	// final target position of joint4 in motor (not DH , same for below defination) 
	m_jnt4TargetPos: LREAL;
	
	// OTG for joint4 motion
	m_trajFilter :FB_secOrdTrajFilter;
	
	// command joint4 position and veloicty in motor for next cycle
	m_cmdJntPos: LREAL;
	m_cmdJntVel: LREAL;
	m_cmdJntAcc: LREAL;

	// PID for joint position
	m_jntPIDCtrl: FB_PID;
	m_jntCtrlTrq: LREAL;
	
END_VAR

METHOD PROTECTED calcJnt6Bias : LREAL
VAR_IN_OUT CONSTANT
	i_masterArm :FB_MasterArm;
END_VAR
IF 1= i_masterArm.armIdx THEN
	calcJnt6Bias :=i_masterArm.curJntPos[6]+PI/2;
ELSE 
	calcJnt6Bias := i_masterArm.curJntPos[6]-PI/2;
END_IF
END_METHOD

// calculate orientation manipulation velocity(in local coordinate)
METHOD calcManipVel : LREAL
VAR_IN_OUT CONSTANT
	i_masterArm :FB_MasterArm;
END_VAR
VAR
	wVelWrd,wVelLocal:Vec3d;
	rotT:Mat3d;
END_VAR
wVelWrd[1]:= i_masterArm.m_curCartLinkTwist[4];
wVelWrd[2]:= i_masterArm.m_curCartLinkTwist[5];
wVelWrd[3]:= i_masterArm.m_curCartLinkTwist[6];

matTranspose(i_masterArm.curCartPose.m_rot, rotT);
matMultiVec(rotT, wVelWrd, wVelLocal);

wVelLocal[3]:=0;
calcManipVel:=norm(wVelLocal);
END_METHOD

METHOD PROTECTED calcNullJaco : Mat4d;
VAR_IN_OUT CONSTANT
	i_masterArm :FB_MasterArm;
END_VAR
VAR
	i,j:INT;
	oriJaco:Mat34;
	oriJt:Mat43;
	oriJJt:Mat3d;
	oriJJtInv:Mat3d;
	oriJPinv:Mat43;
	JpinvJ :Mat4d;
	eye4d :Mat4d := g_eye4d;
END_VAR
// compute pinv of orientation jacobian
FOR i:=1 TO 3 DO
	FOR j:=1 TO 4 DO
		oriJaco[i,j]:=i_masterArm.simJaco[i+3,j+3];
	END_FOR
END_FOR
matTranspose(oriJaco, oriJt);
matMultiply(oriJaco ,oriJt , oriJJt);
invMat3(oriJJt, oriJJtInv);
matMultiply(oriJt, oriJJtInv, oriJPinv);

// calculate nullspace
matMultiply(oriJPinv, oriJaco, JpinvJ);
matSub(eye4d , JpinvJ, calcNullJaco);
END_METHOD

METHOD PROTECTED calcRedunPos : BOOL
VAR_IN_OUT CONSTANT
	i_masterArm :FB_MasterArm;
END_VAR

VAR 
	j6Bias :LREAL;
	curJntPos : Vec7d;
	jnt4LinkPos, jnt4TargetLinkPos :LREAL;
	singScale:LREAL;
END_VAR
// compute desired joint4 link position
// therotically should be link position, but joint controller use motor pos, so here also use motor pos, or will cause other problems
curJntPos :=  i_masterArm.curJntPos;
jnt4LinkPos:=i_masterArm.jnt4MotorToLink(curJntPos[2],curJntPos[3],curJntPos[4]);

// scale track motion near redundant singularity
IF ABS(m_oriNullJaco[1,1])<g_smallNum THEN
	singScale :=0;
ELSE
	singScale := MAX(ABS(m_oriNullJaco[2,1]/m_oriNullJaco[1,1]), ABS(m_oriNullJaco[3,1]/m_oriNullJaco[1,1]));
END_IF
j6Bias := m_jnt6Bias * ABS(singScale);

j6Bias := LIMIT (-m_maxTargetPosStep, j6Bias, m_maxTargetPosStep);
// final target position
jnt4TargetLinkPos := LIMIT(GVL_ArmJointParameters.g_minJntPos[i_masterArm.armIdx,4]+m_jntLimitBuffer, 
			jnt4LinkPos-j6Bias,GVL_ArmJointParameters.g_maxJntPos[i_masterArm.armIdx,4]-m_jntLimitBuffer); 
			
// convert from link position to motor position
m_jnt4TargetPos:=i_masterArm.jnt4LinkToMotor(curJntPos[2], curJntPos[3], jnt4TargetLinkPos);
END_METHOD

METHOD init : BOOL
VAR_IN_OUT CONSTANT
	i_masterArm :FB_MasterArm;
END_VAR
VAR
	currentRatioMotor2Jnt:LREAL;
END_VAR
m_cmdJntPos:=i_masterArm.curJntPos[4];
m_jnt4TargetPos:=m_cmdJntPos;
m_cmdJntVel:=0;

// init controller
currentRatioMotor2Jnt:=GVL_ArmJointParameters.g_motorTrqConst[4]*GVL_ArmJointParameters.g_motorReduction[4]/1000;
m_jntPIDCtrl.init(g_armCtrlCycleTime,m_redunJntKp,m_redunJntKd,m_redunJntKi,
		m_redunJntKiLimit* currentRatioMotor2Jnt,	m_redunJntCtrlLimit*currentRatioMotor2Jnt);

// init OTG
m_trajFilter.init(m_cmdJntPos,m_cmdJntVel,m_jnt4MaxFollowVel,m_jnt4MaxFollowAcc,g_armCtrlCycleTime);
END_METHOD

METHOD run : LREAL
VAR_IN_OUT CONSTANT
	i_masterArm :FB_MasterArm;
END_VAR
VAR_INPUT
	i_followEnable :BOOL;
END_VAR


VAR
	velScale,limitScale:LREAL;
	maxAcc, minDec:LREAL;
	wVel:Vec3d;

END_VAR
// joint 6 deviation from center
m_jnt6Bias := calcJnt6Bias(i_masterArm);

// calculate nullspace jacobian
m_oriNullJaco := calcNullJaco(i_masterArm);

// calculate manipulation angular velocity(exclude roll velocity)
m_curManipWVel := calcManipVel(i_masterArm);

// check if arm is static
m_trackFlag := startTrackCheck(i_masterArm);

// determin target position of joint4
IF i_followEnable THEN
	// update target redundant joint position
	IF  m_trackFlag THEN
		calcRedunPos(i_masterArm);
	ELSE
		// no control in static state
		IF ABS(m_cmdJntPos-m_jnt4TargetPos)< m_joint4TrackTol THEN
			m_jnt4TargetPos := i_masterArm.curJntPos[4];
			m_cmdJntPos :=i_masterArm.curJntPos[4];
			m_cmdJntVel:=0;
			m_jntPIDCtrl.reset();
			m_trajFilter.init(m_cmdJntPos,m_cmdJntVel,m_jnt4MaxFollowVel,m_jnt4MaxFollowAcc,g_armCtrlCycleTime);
		END_IF
	END_IF
END_IF

// scale following acceleration based on manipulation velocity
velScale := LIMIT (0,(ABS(m_curManipWVel)-m_jnt4MinAccVel)/(m_jnt4MaxAccVel-m_jnt4MinAccVel), 1.0);
maxAcc:=(m_jnt4MaxFollowAcc-m_jnt4MinFollowAcc)*velScale+m_jnt4MinFollowAcc;
//minDec:=m_trajFilter.minDec(m_jnt4TargetPos);
//maxAcc := MAX(maxAcc, minDec);

// scale acceleration when approaching limit
//m_accScaleNearLimit:=1;
limitScale := LIMIT(0.0,(ABS(m_jnt6Bias) - m_accScaleBiasLB)/(m_accScaleBiasUB-m_accScaleBiasLB),1.0);
m_accScaleNearLimit := 1+ limitScale * velScale * m_maxAccScaleNearLimit;
maxAcc:=maxAcc*m_accScaleNearLimit;


// run OTG
m_trajFilter.maxV:=m_curManipWVel;
m_trajFilter.maxA:=maxAcc;
m_trajFilter.run(m_jnt4TargetPos, 0.0, o_cmdAcc=>m_cmdJntAcc,o_cmdVel=>m_cmdJntVel, o_cmdPos=>m_cmdJntPos);

// joint position control torque control
m_jntCtrlTrq:=m_jntPIDCtrl.run(m_cmdJntPos,i_masterArm.curJntPos[4], m_cmdJntVel, i_masterArm.curJntVel[4]);

run:=m_jntCtrlTrq;
END_METHOD

METHOD startTrackCheck : BOOL
VAR_IN_OUT CONSTANT
	i_masterArm :FB_MasterArm;
END_VAR
IF (m_curManipWVel> m_staticVelThres AND i_masterArm.m_curLinkVel[6] * m_jnt6Bias > 0)  OR ABS(m_jnt6Bias)> m_staticBiasThres THEN
	startTrackCheck := TRUE;
ELSE
	startTrackCheck :=FALSE;
END_IF
END_METHOD

END_FUNCTION_BLOCK

// ---- FBs_TrajectoryPlanning/OTG/FB_secOrdTrajFilter.TcPOU
// reference: trajectory planning for automatic machines and robots
FUNCTION_BLOCK FB_secOrdTrajFilter
VAR_INPUT
END_VAR
VAR_OUTPUT
END_VAR
VAR
	// command pos and vel from last cycle
	m_cmdPos :LREAL;
	m_cmdVel :LREAL;
	
	// max velocity and acceleration
	m_maxV :LREAL;
	m_maxA :LREAL;
	
	// samping time
	m_Ts :LREAL;
	
	// middle variable
	ek,ek_dot,zk,zk_dot,m,sigma,satSigma :LREAL;

END_VAR

METHOD init : BOOL
VAR_INPUT
	i_curCmdPos : LREAL;
	i_curCmdVel :LREAL;
	i_maxV : LREAL;
	i_maxA :LREAL;
	i_Ts :LREAL;
END_VAR
m_cmdPos:=i_curCmdPos;
m_cmdVel:=i_curCmdVel;
m_maxV :=i_maxV;
m_maxA :=i_maxA;
m_Ts :=i_Ts;
END_METHOD

PROPERTY PUBLIC maxA : LREAL
GET
maxA:=m_maxA;
END_GET
SET
m_maxA :=maxA;
END_SET
END_PROPERTY

PROPERTY PUBLIC maxV : LREAL
GET
maxV:=m_maxV;
END_GET
SET
m_maxV:=maxV;
END_SET
END_PROPERTY

// get minimum deceleration to avoid overshoot
METHOD PUBLIC minDec : LREAL
VAR_INPUT
	i_targetPos : LREAL;
END_VAR

VAR
	dis : LREAL;
END_VAR
dis := i_targetPos-m_cmdPos;
// if target position reverse direciton, there always be a overshoot
IF dis*m_cmdVel <0 THEN
	minDec :=g_smallNum;
	RETURN;
END_IF

dis := MAX(g_smallNum, ABS(dis));
minDec := m_cmdVel *m_cmdVel /(2*dis);
END_METHOD

METHOD run : BOOL
VAR_INPUT
	i_targetPos, i_targetVel :LREAL;
END_VAR

VAR_OUTPUT
	o_cmdAcc, o_cmdVel, o_cmdPos :LREAL;
END_VAR
    ek:=(m_cmdPos-i_targetPos)/m_maxA;
    ek_dot:=(m_cmdVel-i_targetVel)/m_maxA;
    
    zk:=(ek/m_Ts+ek_dot/2)/m_Ts;
    zk_dot:=ek_dot/m_Ts;
    
    m:= floor((1+SQRT(1+8*ABS(zk)))/2);
    sigma:=zk_dot+zk/m+sign(zk)*(m-1)/2;
    satSigma:=MIN(1, MAX(-1,sigma));
    
    o_cmdAcc:=-m_maxA*satSigma*(1+sign(m_cmdVel*sign(sigma)+m_maxV-m_Ts*m_maxA))/2;
    o_cmdVel:=m_cmdVel+o_cmdAcc*m_Ts;
    o_cmdPos:=m_CmdPos+(o_cmdVel+m_cmdVel)*m_Ts/2;
	
	m_cmdVel := o_cmdVel;
	m_cmdPos := o_cmdPos;
END_METHOD

END_FUNCTION_BLOCK

// ---- AgiMaths/MatrixLib/invMat3.TcPOU
FUNCTION invMat3 : bool
VAR_IN_OUT CONSTANT
	mat :Mat3d;
END_VAR
VAR_IN_OUT
	invMat : Mat3d;
END_VAR
VAR
	n:INT:=3;
	m:INT:=1;
	b :ARRAY[1..3] OF LREAL := [3(0)];
	indxc,indxr, ipiv:ARRAY[1..3] OF INT := [3(0)];

	
	i,icol, irow, j,k,l,ll: INT;
	big, dum, pivinv,tmp: LREAL;
END_VAR

invMat := mat;
FOR i:=1 TO n DO   
    big:=0.0;
    FOR j:=1 TO n DO  
        IF (ipiv[j] <> 1) THEN
            FOR k:=1 TO n DO 
                IF (ipiv[k] = 0) THEN
                    IF (ABS(invMat[j,k]) >= big) THEN
                        big:=ABS(invMat[j,k]);
                        irow:=j;
                        icol:=k;
                    END_IF
                END_IF
            END_FOR
        END_IF
    END_FOR
    ipiv[icol]:=ipiv[icol]+1;
    
    IF (irow <> icol) THEN
        FOR l:=1 TO n DO 
            tmp:=invMat[irow,l];
            invMat[irow,l]:=invMat[icol,l];
            invMat[icol,l]:=tmp;
        END_FOR
 (*       FOR  l:=1 TO m DO  
            tmp:=b[irow,l];
            b[irow,l]:=b[icol,l];
            b[icol,l]:=tmp;
        END_FOR*)
    END_IF
	
    indxr[i]:=irow; 
    indxc[i]:=icol;
	
 	IF ABS(invMat[icol,icol]) < g_smallNum THEN  
          invMat3:=FALSE;
		  RETURN;
    END_IF
	
    pivinv:=1.0/invMat[icol,icol];
    invMat[icol,icol]:=1.0;
    FOR l:=1 TO n DO  
        invMat[icol,l] := invMat[icol,l]*pivinv;
    END_FOR
 (*   FOR l:=1 TO m DO 
        b[icol,l] := b[icol,l]*pivinv;
    END_FOR*)
    FOR ll:=1 TO n DO  
        IF (ll <> icol) THEN 
            dum:=invMat[ll,icol];
            invMat[ll,icol]:=0.0;
            FOR l:=1 TO n DO  
                invMat[ll,l]:=invMat[ll,l] - invMat[icol,l]*dum;
            END_FOR
   (*         FOR l:=1 TO m DO  
                b[ll,l]:=b[ll,l] - b[icol,l]*dum;
            END_FOR*)
        END_IF
    END_FOR

END_FOR


FOR l:=n-1 TO 1 BY -1 DO 
    IF (indxr[l] <> indxc[l]) THEN
        FOR k:=1 TO n DO
            tmp:=invMat[k,indxr[l]];
            invMat[k,indxr[l]]:=invMat[k,indxc[l]];
            invMat[k,indxc[l]]:=tmp;
        END_FOR
    END_IF
END_FOR

invMat3:=TRUE;

END_FUNCTION

// ---- AgiMaths/MatrixLib/matSub.TcPOU
// C = A - B;
FUNCTION matSub : BOOL
VAR_IN_OUT CONSTANT
	matA :ARRAY[*,*] OF LREAL;
	matB :ARRAY[*,*] OF LREAL;
END_VAR

VAR_IN_OUT 
	matC :ARRAY[*,*] OF LREAL;
END_VAR

VAR
	m,n :DINT;
	i,j, k :DINT;
 
END_VAR

m:=UPPER_BOUND(matC,1);
n:= UPPER_BOUND(matC,2);
ASSERT(UPPER_BOUND(matA,1)=m);
ASSERT(UPPER_BOUND(matA,2)=n);
ASSERT(UPPER_BOUND(matB,1)=m);
ASSERT(UPPER_BOUND(matB,2)=n);
FOR i:=1 TO m DO
	FOR j:=1 TO n DO
		matC[i,j]:=matA[i,j]-matB[i,j];
	END_FOR
END_FOR

END_FUNCTION

// ---- FBs_BasicControllers/FB_boundaryForceFeedback.TcPOU
FUNCTION_BLOCK FB_boundaryForceFeedback
VAR_INPUT
END_VAR
VAR_OUTPUT
END_VAR

VAR
	// force control parameters in local tip coordinate
//	m_oriKp :Vec3d :=[1, 1, 0.5];
//	m_oriKd :Vec3d :=[0.04,0.04, 0.01];
	m_oriKp :Vec3d :=[0.2, 0.2, 0.1];
	m_oriKd :Vec3d :=[0.02,0.02, 0.005];

	m_oriCartTrq,m_oriCartTrqLocal :Vec3d;
	
	m_posKp :LREAL := 200;
	m_posKd :LREAL := 10;
	m_posCartForce:Vec3d;
	
	
END_VAR

METHOD run : Vec7d

VAR_IN_OUT CONSTANT
	i_slaveIdx :INT;
	i_shoulderPose :ST_Frame;
	i_masterArm :FB_MasterArm;
	i_slaveStatus :ST_SlaveStatus;
END_VAR

VAR
	posErrInScope, oriErrInScope:Vec3d;
	posErr, oriErr:Vec3d;
	posErrLocal, oriErrLocal :Vec3d;
	vel, velLocal, wVel,wVelLocal :Vec3d;
	oriErrAxis, wVelProj :Vec3d;
	rotInv :Mat3d;
	oriJaco, oriJacoT :Mat3d;
	oriJntTrq :Vec3d;
	
	i,j:INT;
	posErrAxis, velProj :Vec3d;
	posJaco, posJacoT :Mat3d;
	posJntTrq :Vec3d;
	
	trqScale :LREAL;
END_VAR
run:=g_zeroVec7d;

FOR i:=1 TO 3 DO
	posErrInScope[i]:= -i_slaveStatus.m_masterSlavePoseError[i_slaveIdx][i];
	oriErrInScope[i]:= -i_slaveStatus.m_masterSlavePoseError[i_slaveIdx][i+3];
	vel[i]:=i_masterArm.curCartTwist[i];
	wVel[i]:=i_masterArm.curCartTwist[i+3];
END_FOR

// calculate pose error in shoulder coordinate
matTranspose(i_shoulderPose.m_rot, rotInv);
matMultiVec(rotInv, posErrInScope, posErr);
matMultiVec(rotInv, oriErrInScope, oriErr);
// ################### 	force  #########################
// add threshold
IF norm(posErr) > g_smallNum THEN
	// project error in tip coordinate
	matTranspose(i_masterArm.curCartPose.m_rot, rotInv);
	matMultiVec(rotInv, posErr, posErrLocal);
	matMultiVec(rotInv, oriErr, oriErrLocal);
	matMultiVec(rotInv, vel, velLocal);
	matMultiVec(rotInv, wVel, wVelLocal);
	
	// compute velocity in error direction
	posErrAxis := posErr;
	normalize(posErrAxis);
	vecMultiNum(posErrAxis, vecDot(vel, posErrAxis), velProj);
	
	// compute local cartesion torque
	FOR i:=1 TO 3 DO
		m_posCartForce[i]:= m_posKp * posErr[i]-m_posKd*velProj[i];
	END_FOR
	
	// compute joint space torque
	FOR i :=1 TO  3 DO
		FOR j:=1 TO 3 DO
			posJaco[i,j]:= i_masterArm.jaco[i,j];
		END_FOR
	END_FOR
	matTranspose(posJaco, posJacoT);
	matMultiVec(posJacoT, m_posCartForce, posJntTrq);
	
	// scale joint troque
	trqScale := 1;
	FOR i:=1 TO 3 DO 
		trqScale:=MAX(trqScale, ABS(posJntTrq[i]/GVL_ArmJointParameters.g_jntMaxTrq[i]));
	END_FOR
	
	run[1]:=posJntTrq[1]/trqScale;
	run[2]:=posJntTrq[2]/trqScale;
	run[3]:=posJntTrq[3]/trqScale;
END_IF


// ###################  torque #########################
// add threshold
IF norm(oriErr) > g_smallNum THEN
	// project error in tip coordinate
	matTranspose(i_masterArm.curCartPose.m_rot, rotInv);
	matMultiVec(rotInv, posErr, posErrLocal);
	matMultiVec(rotInv, oriErr, oriErrLocal);
	matMultiVec(rotInv, vel, velLocal);
	matMultiVec(rotInv, wVel, wVelLocal);
	
	// compute velocity in error direction
	oriErrAxis := oriErrLocal;
	normalize(oriErrAxis);
	vecMultiNum(oriErrAxis, vecDot(wVelLocal, oriErrAxis), wVelProj);
	
	// compute local cartesion torque
	FOR i:=1 TO 3 DO
		m_oriCartTrqLocal[i]:= m_oriKp[i] * oriErrLocal[i]-m_oriKd[i]*wVelProj[i];
	END_FOR
	
	// project torque back to shoulder coordinate
	matMultiVec(i_masterArm.curCartPose.m_rot, m_oriCartTrqLocal, m_oriCartTrq);
	
	// compute joint space torque
	// for simplicity, we current only use last 3 joint for torque feedback
	FOR i :=1 TO  3 DO
		FOR j:=1 TO 3 DO
			oriJaco[i,j]:= i_masterArm.jaco[i+3,j+4];
		END_FOR
	END_FOR
	matTranspose(oriJaco, oriJacoT);
	matMultiVec(oriJacoT, m_oriCartTrq, oriJntTrq);
	
	// scale joint troque
	trqScale := 1;
	FOR i:=1 TO 3 DO 
		trqScale:=MAX(trqScale, ABS(oriJntTrq[i]/GVL_ArmJointParameters.g_jntMaxTrq[i+4]));
	END_FOR
	
	run[5]:=oriJntTrq[1]/trqScale;
	run[6]:=oriJntTrq[2]/trqScale;
	run[7]:=oriJntTrq[3]/trqScale;
END_IF
END_METHOD

END_FUNCTION_BLOCK

// ---- AgiMaths/MatrixLib/vecDot.TcPOU
// vecB=VecA*num
FUNCTION vecDot : LREAL
VAR_IN_OUT CONSTANT
	vecA :ARRAY[*] OF LREAL;
	vecB :ARRAY[*] OF LREAL;
END_VAR

VAR
	m :DINT;
	i :DINT;
END_VAR

m:=UPPER_BOUND(vecA,1);
ASSERT(UPPER_BOUND(VecB,1)=m);

vecDot :=0;
FOR i:=1 TO m DO
	vecDot := vecDot + vecA[i]*vecB[i];
END_FOR

END_FUNCTION

// ---- AgiMaths/MatrixLib/vecSelfMultiNum.TcPOU
// vecA*=num
FUNCTION vecSelfMultiNum : BOOL
VAR_IN_OUT 
	vecA :ARRAY[*] OF LREAL;
END_VAR

VAR_INPUT
	num :LREAL;
END_VAR

VAR
	m :DINT;
	i :DINT;
 
END_VAR

m:=UPPER_BOUND(vecA,1);

FOR i:=1 TO m DO
		vecA[i]:=num*vecA[i];
END_FOR

END_FUNCTION

// ---- FBs_StateControllers/FB_StateCtrlClutch.TcPOU
// Brief: Master Arm Clutch
FUNCTION_BLOCK PUBLIC FB_StateCtrlClutch EXTENDS FB_MasterArmCtrlBase
VAR_INPUT
END_VAR
VAR_OUTPUT
END_VAR
VAR
	// orientation tracking parameters
	m_rotTrackKp : LREAL := 200;
	m_maxTrackVel :LREAL := PI;
	
	// redundant control parameters
	m_jnt4AdjustKp : LREAL :=10;
	m_jnt4MaxVel :LREAL :=pi/3 ;
	m_linearVelLb :LREAL := 0.02;
	m_linearVelUb :LREAL :=0.1;	
	
END_VAR

// override this function in each exact controller
METHOD PROTECTED calcCmdJntPos : BOOL

VAR_IN_OUT CONSTANT
	i_slaveIdx :INT;
	i_shoulderPose :ST_Frame;
	i_masterArm :FB_MasterArm;
	i_slaveStatus :ST_SlaveStatus;
END_VAR
var 
	i,j : INT;
	rotT,rotErr:Mat3d;
	angle : LREAL;
	axis,localAxis :Vec3d;
	oriJaco:Mat34;
	oriJt:Mat43;
	oriJJt:Mat3d;
	oriJJtInv:Mat3d;
	oriJPinv:Mat43;
	cartTrackVel:Vec3d;
	jntTrackVel:Vec4d;
	JpinvJ, nullJ:Mat4d;
	eye4d :Mat4d := g_eye4d;
	redunCtrlVel :Vec4d;
	jnt4TrackVel :LREAL;
	
END_VAR
// TODO: use matched slave arm orientation as target, 
//	and transform from view coordinate to arm coordinate 

// first three joints is passive control
FOR i:=1 TO 3 DO 
	m_cmdJntPos[i]:=i_masterArm.curJntPos[i];
	m_cmdJntVel[i]:=i_masterArm.curJntVel[i];
END_FOR

// compute cartesian tracking velocity
matTranspose(i_masterArm.simCartPose.m_rot, rotT);
matMultiply(rotT, m_cmdCartPose.m_rot, rotErr);
rot2AngAxis(rotErr, angle=>angle,axis=>localAxis);
matMultiVec(i_masterArm.simCartPose.m_rot, localAxis, axis);
vecMultiNum(axis, LIMIT(-m_maxTrackVel, angle*m_rotTrackKp, m_maxTrackVel), cartTrackVel);

// compute pinv of orientation jacobian
FOR i:=1 TO 3 DO
	FOR j:=1 TO 4 DO
		oriJaco[i,j]:=i_masterArm.simJaco[i+3,j+3];
	END_FOR
END_FOR
matTranspose(oriJaco, oriJt);
matMultiply(oriJaco ,oriJt , oriJJt);
invMat3(oriJJt, oriJJtInv);
matMultiply(oriJt, oriJJtInv, oriJPinv);
matMultiVec(oriJpinv, cartTrackVel, jntTrackVel);

// calculate nullspace
matMultiply(oriJPinv, oriJaco, JpinvJ);
matSub(eye4d , JpinvJ, nullJ);

// redundant velocity
jnt4TrackVel:=calcRedunVel(i_masterArm);
redunCtrlVel[1]:=nullJ[1,1]*jnt4TrackVel;
redunCtrlVel[2]:=nullJ[2,1]*jnt4TrackVel;
redunCtrlVel[3]:=nullJ[3,1]*jnt4TrackVel;
redunCtrlVel[4]:=nullJ[4,1]*jnt4TrackVel;

// update final command joint position and velocity
FOR i :=1 TO 4 DO 
//	m_cmdJntVel[i+3]:=jntTrackVel[i];
	m_cmdJntVel[i+3]:=jntTrackVel[i]+redunCtrlVel[i];
	m_cmdJntPos[i+3]:=m_cmdJntPos[i+3]+m_cmdJntVel[i+3]*g_armCtrlCycleTime;
END_FOR
END_METHOD

METHOD PROTECTED calcRedunVel : LREAL
VAR_IN_OUT CONSTANT
	i_masterArm :FB_MasterArm;
END_VAR

VAR 
	j6Bias,j5Bias :LREAL;
	velScale :LREAL;
	linearVel :Vec3d;
	curJntPos : Vec7d;
	jnt4LinkPos :LREAL;
END_VAR
// compute desired joint4 link position
curJntPos :=  i_masterArm.cmdJntPos;
jnt4LinkPos:=i_masterArm.jnt4MotorToLink(curJntPos[2],curJntPos[3],curJntPos[4]);
IF 1= i_masterArm.armIdx THEN
	j6Bias :=curJntPos[6]+PI/2;
ELSE 
	j6Bias := curJntPos[6]-PI/2;
END_IF

// scale based on joint5 position
j5Bias :=  LIMIT (0, ABS(curJntPos[5] -pi), pi/2);
j6Bias := j6Bias * ABS(COS(j5Bias));

// scale based on linear velocity
linearVel[1]:=i_masterArm.curCartTwist[1];
linearVel[2]:=i_masterArm.curCartTwist[2];
linearVel[3]:=i_masterArm.curCartTwist[3];
velScale :=LIMIT(0, (norm(linearVel)-m_linearVelLb)/(m_linearVelUb-m_linearVelLb),1.0);


calcRedunVel := LIMIT(-m_jnt4MaxVel, -j6Bias * m_jnt4AdjustKp * velScale ,m_jnt4MaxVel);

// joint limit
IF (calcRedunVel > 0 AND jnt4LinkPos+calcRedunVel * g_armCtrlCycleTime > GVL_ArmJointParameters.g_maxJntPos[i_masterArm.armIdx,4])
	 OR ( calcRedunVel <0 AND  jnt4LinkPos +calcRedunVel * g_armCtrlCycleTime< GVL_ArmJointParameters.g_minJntPos[i_masterArm.armIdx,4]) THEN
	 calcRedunVel :=0;
END_IF
END_METHOD

METHOD PUBLIC init : BOOL
VAR_IN_OUT CONSTANT
	i_masterArm	:FB_MasterArm;
END_VAR
VAR_IN_OUT 
	r_masterArmCtrlCmd :ST_ArmCtrlCmds;
END_VAR

VAR
	i:INT;
END_VAR
SUPER^.Init(i_masterArm,r_masterArmCtrlCmd);

m_jntOPMode[1] := DriverOPMode_Trq;
m_jntOPMode[2] := DriverOPMode_Trq;
m_jntOPMode[3] := DriverOPMode_Trq;
m_jntOPMode[4] := DriverOPMode_PosTrq;
m_jntOPMode[5] := DriverOPMode_PosTrq;
m_jntOPMode[6] := DriverOPMode_PosTrq;
m_jntOPMode[7] := DriverOPMode_PosTrq;

// update commands to arm
copyCmds(r_masterArmCtrlCmd);
END_METHOD

END_FUNCTION_BLOCK

// ---- FBs_StateControllers/FB_StateCtrlEndoscope.TcPOU
// Brief: Master Arm Endoscope Control
FUNCTION_BLOCK PUBLIC FB_StateCtrlEndoscope EXTENDS FB_MasterArmCtrlBase
VAR_INPUT
END_VAR
VAR_OUTPUT
END_VAR
VAR
	// enter endoscope control for the first time
	m_firstIn :BOOL := TRUE;
	
	//arm force control in base coordinate
	m_impCtrlInBase:BOOL;
	
	// force control parameters in base coordinate
	m_kpBase:Vec6d:=[1,1,1,1,1,1];
	m_kdBase:Vec6d:=[0.01,0.01,0.01,0.01,0.01,0.01];
	
	//endoscope motion scale
	m_endoMotionScale:LREAL:=1;
	
	// force control parameters in tcp coordinate
	m_kpTcp:Vec6d:=[100,100,100,1,1,0.5];
	m_kdTcp:Vec6d:=[1,1,1,0.04,0.04,0.01]; //[5,5,5,0.04,0.04,0.01];
	
	//joint 6 KP/KD
	m_Kp6:LREAL:=1.0; //1
	m_Kd6:LREAL:=0.01; //0.01
	
	//expected joint 6 position
	m_ExpJ6Pos:LREAL;
	
	//time
	m_t:LREAL;	
END_VAR

// override this function in each exact controller
METHOD PROTECTED calcCmdJntPos : BOOL

VAR_IN_OUT CONSTANT
	i_slaveIdx :INT;
	i_shoulderPose :ST_Frame;
	i_masterArm :FB_MasterArm;
	i_slaveStatus :ST_SlaveStatus;
END_VAR
VAR 

END_VAR
m_cmdJntPos:=i_masterArm.curJntPos;
m_cmdJntVel:=i_masterArm.curJntVel;
m_cmdCartPose:=i_masterArm.curCartPose;
END_METHOD

// override this function in each exact controller
METHOD PROTECTED calcCmdJntTrq : BOOL

VAR_IN_OUT CONSTANT
	i_slaveIdx :INT;
	i_shoulderPose :ST_Frame;
	i_masterArm :FB_MasterArm;
	i_slaveStatus :ST_SlaveStatus;
END_VAR

VAR	
	i:INT;
	
	//position variables
	masterPos,slavePos:ST_Frame;
	masterPosFirst,slavePosFirst:ST_Frame;
	ArmTarPos:ST_Frame;
	posInc:Vec3d;		
	tmpMat3d : Mat3d;
	rotInv:Mat3d;
	
	//velocity variables
	vel, velLocal, wVel,wVelLocal :Vec3d;
	spatialVel,spatialVelInTcp:Vec6d;
	
	//force variables
	spatialForceP1,spatialForceP2:Vec3d;	
	spatialForceP1Base,spatialForceP2Base:Vec3d;		
	spatialForTcp,spatialForBase,spatialForTemp:Vec7d;
	
	//joint torque variables
	simJaco:Mat67;
	JacoT :Mat76;	
	jntTorVec:Vec7d;
	dynaNullspace:Mat7d;	
	TorqueNullSpace:Vec7d; //joint torque for null space
	jntOptTor:LREAL; //joint 6 optimization torque
	jntTorqueSum:Vec7d;		
	jntImpTor:Vec7d;
	
	//master arm posture error variables
	posErr,posErrInBase,posErrInTcp:Vec3d;
	rotErr :Mat3d;
	errAngle : LREAL;
	errAxisLocal, errAxis,errAxis2,errAxisInBase,errAxisInTcp :Vec3d;
	masterPoseError,masterPoseErrorInTcp :Vec6d;
END_VAR

//determine slave arm space position relative to endoscope
masterPos:=transform(i_shoulderPose,i_masterArm.simCartPose);
slavePos:=i_slaveStatus.m_curArmPose[i_slaveIdx];

//system parameters initial
IF (m_firstIn=TRUE) THEN
	m_firstIn:=FALSE;
	masterPosFirst:=masterPos;
	slavePosFirst:=slavePos;	
	m_ExpJ6Pos:=i_masterArm.curJntPos[6];	
END_IF

m_t:=m_t+g_armCtrlCycleTime;
IF (m_t<=0.050) THEN
	m_firstIn:=TRUE;
	RETURN;	
END_IF




//calculating slave arm position incresement，and determine master arm space position and posture
vecSub(slavePos.m_pos,slavePosFirst.m_pos,posInc);
vecMultiNum(posInc,1.0/m_endoMotionScale,posInc);
vecAdd(posInc,masterPosFirst.m_pos,ArmTarPos.m_pos);
ArmTarPos.m_rot:=slavePos.m_rot;



//calculating master arm position error and postrue error
vecSub(ArmTarPos.m_pos, masterPos.m_pos, PosErr);
matTranspose(masterPos.m_rot, tmpMat3d);
matMultiply(tmpMat3d, ArmTarPos.m_rot, rotErr);
rot2AngAxis(rotErr, angle=>errAngle, axis=>errAxisLocal);
matMultiVec(masterPos.m_rot, errAxisLocal, errAxis);



//transform the error to arm base coordinate
matTranspose(i_shoulderPose.m_rot,tmpMat3d); //transform matrix from eye to base
matMultiVec(tmpMat3d, PosErr,posErrInBase);
matMultiVec(tmpMat3d, errAxis,errAxis2);
vecMultiNum(errAxis2,errAngle,errAxisInBase);
FOR i:=1 TO 3 BY 1 DO
	masterPoseError[i]:=posErrInBase[i];
	masterPoseError[i+3]:=errAxisInBase[i];
END_FOR



//transform the error to TCP coordinate
matTranspose(i_masterArm.curCartPose.m_rot, rotInv);
matMultiVec(rotInv, posErrInBase, posErrInTcp);
matMultiVec(rotInv, errAxisInBase, errAxisInTcp);
FOR i:=1 TO 3 BY 1 DO
	masterPoseErrorInTcp[i]:=posErrInTcp[i];
	masterPoseErrorInTcp[i+3]:=errAxisInTcp[i];
END_FOR



//determine master arm space velocity in base coordinate
FOR i:=1 TO 3 DO
	vel[i]:=i_masterArm.curCartTwist[i];
	wVel[i]:=i_masterArm.curCartTwist[i+3];
	spatialVel[i]:=vel[i];
	spatialVel[i+3]:=wVel[i];
END_FOR



//transform master arm space velocity to tcp coordinate
matMultiVec(rotInv, vel, velLocal);
matMultiVec(rotInv, wVel, wVelLocal);
FOR i:=1 TO 3 DO
	spatialVelInTcp[i]:=velLocal[i];
	spatialVelInTcp[i+3]:=wVelLocal[i];
END_FOR



//Jacobian matrix
simJaco:=i_masterArm.Jaco;



//Based on the above pose deviation values, input them into the impedance control equation and derive the impedance joint torque value
IF (m_impCtrlInBase=TRUE) THEN
	FOR i:=1 TO 6 BY 1 DO
		spatialForBase[i]:=m_kpBase[i]*masterPoseError[i]-m_kdBase[i]*spatialVel[i]; //(-1)*err*(-1)=err
	END_FOR
	matMultiVec(i_masterArm.m_lambda, spatialForBase, spatialForTemp);
	matTranspose(simJaco,JacoT);
	matMultiVec(JacoT, spatialForTemp, jntImpTor);	
	
ELSE // impedance control in tcp coordinate
	FOR i:=1 TO 6 BY 1 DO
		spatialForTcp[i]:=m_kpTcp[i]*masterPoseErrorInTcp[i]-m_kdTcp[i]*spatialVelInTcp[i];
	END_FOR
	
	//Splitting spatial forces into two parts
	FOR i:=1 TO 3 BY 1 DO
		spatialForceP1[i]:=spatialForTcp[i];
		spatialForceP2[i]:=spatialForTcp[i+3];
	END_FOR
	
	// project torque back to base coordinate	
	matMultiVec(i_masterArm.curCartPose.m_rot, spatialForceP1, spatialForceP1Base);	
	matMultiVec(i_masterArm.curCartPose.m_rot, spatialForceP2, spatialForceP2Base);	
	
	FOR i:=1 TO 3 BY 1 DO
		spatialForBase[i]:=spatialForceP1Base[i];
		spatialForBase[i+3]:=spatialForceP2Base[i];
	END_FOR
	
	//compute joint space torque
	matTranspose(simJaco,JacoT);
	matMultiVec(JacoT, spatialForBase, jntImpTor);	
END_IF




//To ensure that joint 6 is in the appropriate position, a single joint impedance controller is constructed
jntOptTor:=m_Kp6*(m_ExpJ6Pos-i_masterArm.curJntPos[6])-m_Kd6*i_masterArm.curJntVel[6];
(*
//Project the torque of joint 6 onto null space
jntTorVec[6]:=jntOptTor;
dynaNullspace:=i_masterArm.dynaNullspace;
matMultiVec(dynaNullspace, jntTorVec, TorqueNullSpace);	

//Calculate the sum of impedance control torque and zero space torque
vecAdd(jntImpTor,TorqueNullSpace,jntTorqueSum);
m_cmdJntTrq:=jntTorqueSum;
*)
m_cmdJntTrq:=jntImpTor;
m_cmdJntTrq[6]:=jntOptTor;
END_METHOD

// override this function in each exact controller
// NOTICE: set joint control mode here, and do some initialization if needed
METHOD PUBLIC init : BOOL
VAR_IN_OUT CONSTANT
	i_masterArm	:FB_MasterArm;
END_VAR
VAR_IN_OUT 
	r_masterArmCtrlCmd :ST_ArmCtrlCmds;
END_VAR

SUPER^.Init(i_masterArm,r_masterArmCtrlCmd);

m_jntOPMode[1] := DriverOPMode_Trq;
m_jntOPMode[2] := DriverOPMode_Trq;
m_jntOPMode[3] := DriverOPMode_Trq;
m_jntOPMode[4] := DriverOPMode_Trq;
m_jntOPMode[5] := DriverOPMode_Trq;
m_jntOPMode[6] := DriverOPMode_Trq;
m_jntOPMode[7] := DriverOPMode_Trq;

m_firstIn:=TRUE;
m_t:=0;

// update commands to arm
copyCmds(r_masterArmCtrlCmd);
END_METHOD

METHOD relativeAngle : bool
VAR_INPUT
	armId:INT;
	x:LREAL;
	y:LREAL;
END_VAR

VAR_OUTPUT
	angle:LREAL;
END_VAR

VAR
	
END_VAR


angle:=atan2(y,x);
IF (armId=1) AND (angle<0) THEN
	angle:=angle+2*pi;
END_IF
END_METHOD

END_FUNCTION_BLOCK

// ---- AgiMaths/Frames/transform.TcPOU
FUNCTION transform : ST_Frame
VAR_IN_OUT CONSTANT
	i_frame1 :ST_Frame;
	i_frame2 :ST_Frame;
END_VAR
VAR
END_VAR

matMultiply(i_frame1.m_rot, i_frame2.m_rot, transform.m_rot);
matMultiVec(i_frame1.m_rot, i_frame2.m_pos,transform.m_pos );
vecAdd(transform.m_pos,i_frame1.m_pos,transform.m_pos);

END_FUNCTION

// ---- FBs_StateControllers/FB_StateCtrlCart.TcPOU
// Brief: Master Arm Cart Control
FUNCTION_BLOCK PUBLIC FB_StateCtrlCart EXTENDS FB_MasterArmCtrlBase
VAR_INPUT
END_VAR
VAR_OUTPUT
END_VAR
VAR
END_VAR

METHOD PUBLIC init : BOOL
VAR_IN_OUT CONSTANT
	i_masterArm	:FB_MasterArm;
END_VAR
VAR_IN_OUT 
	r_masterArmCtrlCmd :ST_ArmCtrlCmds;
END_VAR
// check if to hold the command joint position unchanged
m_holdLastCmds := checkToHoldLastCmds(i_masterArm);

// init
SUPER^.Init(i_masterArm,r_masterArmCtrlCmd);
END_METHOD

END_FUNCTION_BLOCK

// ---- FBs_StateControllers/FB_StateCtrlGraCali.TcPOU
// Brief: Master Arm Home Posture
FUNCTION_BLOCK PUBLIC FB_StateCtrlGraCali EXTENDS FB_MasterArmCtrlBase
VAR_INPUT
END_VAR
VAR_OUTPUT
END_VAR
VAR CONSTANT
	m_caliMotionSegs :INT :=6;	
END_VAR
VAR
	// cali trajectory
	m_leftGraCaliTraj :ARRAY [1..m_caliMotionSegs, 1..g_mJntNum] OF LREAL:=
		// first calibration traj
		[0,  -60*g_deg2Rad,    0.0,  -195*g_deg2Rad,  270*g_deg2rad,  -60*g_deg2rad, 0.0 , 
		 0, -120*g_deg2rad,   0.0,  -165*g_deg2rad,   90*g_deg2rad,  -120*g_deg2rad,  0,
		 0,  -60*g_deg2Rad,    0.0,  -195*g_deg2Rad,  270*g_deg2rad,  -60*g_deg2rad, 0.0 , 
		// second calibration traj
		 0.0,  -75*g_deg2Rad,   30*g_deg2Rad,  -195*g_deg2Rad,  180*g_deg2Rad,  -90*g_deg2Rad,    0,
		 0.0,  -105*g_deg2Rad,  -30*g_deg2Rad, -165*g_deg2Rad,  180*g_deg2Rad,  -90*g_deg2Rad,     0,
		0.0,  -75*g_deg2Rad,   30*g_deg2Rad,  -195*g_deg2Rad,  180*g_deg2Rad,  -90*g_deg2Rad,    0];
		
	m_rightGraCaliTraj :ARRAY [1..m_caliMotionSegs, 1..g_mJntNum] OF LREAL:=
		// first calibration traj
		[0,   -60*g_deg2Rad,    0.0,   75*g_deg2Rad,   90*g_deg2Rad,   60*g_deg2Rad,  0.0,
		 0.0,  -120*g_deg2Rad,  0.0,  -75*g_deg2Rad,  270*g_deg2Rad,  120*g_deg2Rad,  0.0,
		 0,   -60*g_deg2Rad,    0.0,   75*g_deg2Rad,   90*g_deg2Rad,   60*g_deg2Rad,  0.0,
		// second calibration traj
		 0.0,  -75*g_deg2Rad,   30*g_deg2Rad,  -15*g_deg2Rad,  180*g_deg2Rad,   90*g_deg2Rad,    0,
		 0.0, -105*g_deg2Rad,  -30*g_deg2Rad,   15*g_deg2Rad,  180*g_deg2Rad,   90*g_deg2Rad,    0,
		 0.0,  -75*g_deg2Rad,   30*g_deg2Rad,  -15*g_deg2Rad,  180*g_deg2Rad,   90*g_deg2Rad,    0];
	

	m_transMaxjntVel:Vec7d:=[7(30*g_deg2rad)];
	m_caliMaxjntVel:Vec7d:=[7(3.0*g_deg2rad)];
	m_caliMaxjntAcc:Vec7d:=[7(1.0)];
	m_caliMaxjntJerk:Vec7d:=[7(2.0)];
	
	m_caliTrajIdx: INT := 1;
	m_caliPlanner: ARRAY[1..m_caliMotionSegs] OF FB_TrajMoveJ;
	
	
END_VAR

// override this function in each exact controller
METHOD PROTECTED calcCmdJntPos : BOOL

VAR_IN_OUT CONSTANT
	i_slaveIdx :INT;
	i_shoulderPose :ST_Frame;
	i_masterArm :FB_MasterArm;
	i_slaveStatus :ST_SlaveStatus;
END_VAR
VAR 
	i :INT;
	curJntVel :Vec7d;
END_VAR
// check if planner is ready
IF m_caliPlanner[m_caliTrajIdx].isGene = FALSE THEN
	calcCmdJntPos:=FALSE;
	RETURN;
END_IF

// traj plan
calcCmdJntPos :=m_caliPlanner[m_caliTrajIdx].evaluate(m_timePeriod, jntPos=> m_cmdJntPos, jntVel=>m_cmdJntVel, jntAcc=> m_cmdJntAcc);

// check if to transit to next segment
curJntVel :=i_masterArm.curJntVel;
IF(m_timePeriod > m_caliPlanner[m_caliTrajIdx].duration  AND norm(curJntVel)<7*g_jntStaticVelThres) THEN
	m_caliTrajIdx:=m_caliTrajIdx+1;
	m_timePeriod:=0;
END_IF

// check if to terminated
IF(m_caliTrajIdx > m_caliMotionSegs) THEN
	m_isFinished:=TRUE;
END_IF
END_METHOD

METHOD PUBLIC init : BOOL
VAR_IN_OUT CONSTANT
	i_masterArm	:FB_MasterArm;
END_VAR
VAR_IN_OUT 
	r_masterArmCtrlCmd :ST_ArmCtrlCmds;
END_VAR

VAR
	i,j :INT;
	startJntPos,endJntPos ,maxVel :Vec7d;
	
	
	
END_VAR
SUPER^.Init(i_masterArm,r_masterArmCtrlCmd);
m_caliTrajIdx :=1;

FOR i:=1 TO m_caliMotionSegs DO
	IF i=1 OR i = 4 THEN
		maxVel := m_transMaxjntVel;
	ELSE
		maxVel := m_caliMaxjntVel;
	END_IF
	
	IF i_masterArm.armIdx=1 THEN
		FOR j:=1 TO 7 DO 
			endJntPos[j]:=m_leftGraCaliTraj[i,j];
			IF i =1 THEN
				startJntPos[j]:=i_masterArm.curJntPos[j];
			ELSE
				startJntPos[j]:=m_leftGraCaliTraj[i-1,j];
			END_IF
		END_FOR
	ELSE
		FOR j:=1 TO 7 DO 
			endJntPos[j]:=m_rightGraCaliTraj[i,j];
			IF i =1 THEN
				startJntPos[j]:=i_masterArm.curJntPos[j];
			ELSE
				startJntPos[j]:=m_rightGraCaliTraj[i-1,j];
			END_IF
		END_FOR
	END_IF
	
	m_caliPlanner[i].init(startJntPos,endJntPos,maxVel, m_caliMaxJntAcc, m_caliMaxJntAcc);
END_FOR


// update commands to arm
copyCmds(r_masterArmCtrlCmd);
END_METHOD

END_FUNCTION_BLOCK

// ---- FBs_StateControllers/FB_StateCtrlTest.TcPOU
// Brief: Master Arm Test
FUNCTION_BLOCK PUBLIC FB_StateCtrlTest EXTENDS FB_MasterArmCtrlBase
VAR_INPUT
END_VAR
VAR_OUTPUT
END_VAR
VAR
	// ################ variables for single DH  joint test ##################
	m_freqTestFlag :BOOL:=FALSE;
	m_initJntPos :Vec7d;
	m_jntMotionFreq :Vec7d :=[0.2, 0.2, 0.1, 4(0.1)];
	m_jntMotionRange :Vec7d :=[pi/6, pi/6, 0.1, 4(pi/6)];
	m_testJntIdx :INT :=1;
	
	m_stepTestFlag :BOOL :=FALSE;
	m_jntStep : LREAL := 5*g_deg2Rad;
	
END_VAR

METHOD PROTECTED calcCmdJntPos : BOOL
VAR_IN_OUT CONSTANT
	i_slaveIdx :INT;
	i_shoulderPose :ST_Frame;
	i_masterArm :FB_MasterArm;
	i_slaveStatus :ST_SlaveStatus;
END_VAR

VAR 
	i:INT :=0;
	errThres :LREAL;
	m_masterGripAngle: INT;
END_VAR
// Just for joint controller test
IF m_testJntIdx >=1 AND m_testJntIdx <=7 THEN
	IF m_freqTestFlag THEN 
		m_cmdJntPos[m_testJntIdx]:=m_initJntPos[m_testJntIdx]+m_jntMotionRange[m_testJntIdx]/2
										+0.5*m_jntMotionRange[m_testJntIdx]*SIN(2*pi*m_jntMotionFreq[m_testJntIdx]*m_timePeriod-pi/2);
		m_cmdJntVel[m_testJntIdx]:=0.5*m_jntMotionRange[m_testJntIdx]*2*pi*m_jntMotionFreq[m_testJntIdx]*COS(2*pi*m_jntMotionFreq[m_testJntIdx]*m_timePeriod-pi/2);
	ELSIF m_stepTestFlag THEN
		m_cmdJntPos[m_testJntIdx]:=m_initJntPos[m_testJntIdx]+m_jntStep;
		m_cmdJntVel[m_testJntIdx]:=0;
	ELSE
		m_timePeriod:=0;
	END_IF
	
END_IF


FOR i:=1 TO 3 DO 
		errThres :=5*g_deg2rad;
	IF ABS(m_cmdJntPos[i]-i_masterArm.curJntPos[i])>errThres THEN
		m_isFinished:=TRUE;
	END_IF
	
END_FOR
END_METHOD

METHOD PUBLIC init : BOOL
VAR_IN_OUT CONSTANT
	i_masterArm	:FB_MasterArm;
END_VAR
VAR_IN_OUT 
	r_masterArmCtrlCmd :ST_ArmCtrlCmds;
END_VAR
// check if to hold the command joint position unchanged
m_holdLastCmds := checkToHoldLastCmds(i_masterArm);

// init
SUPER^.Init(i_masterArm,r_masterArmCtrlCmd);

m_initJntPos := i_masterArm.curJntPos;

// update commands to arm
copyCmds(r_masterArmCtrlCmd);
END_METHOD

END_FUNCTION_BLOCK

// ---- FBs_StateControllers/FB_StateCtrlDisable.TcPOU
// Brief: Master Arm Error Hold
FUNCTION_BLOCK PUBLIC FB_StateCtrlDisable EXTENDS FB_MasterArmCtrlBase
VAR_INPUT
END_VAR
VAR_OUTPUT
END_VAR
VAR
END_VAR

// override this function in each exact controller
METHOD PROTECTED calcCmdJntPos : BOOL

VAR_IN_OUT CONSTANT
	i_slaveIdx :INT;
	i_shoulderPose :ST_Frame;
	i_masterArm :FB_MasterArm;
	i_slaveStatus :ST_SlaveStatus;
END_VAR
var 
	i,j : INT;

	
END_VAR
m_cmdJntPos:= i_masterArm.curJntPos;
m_cmdJntVel := g_zeroVec7d;
END_METHOD

METHOD PUBLIC init : BOOL
VAR_IN_OUT CONSTANT
	i_masterArm	:FB_MasterArm;
END_VAR
VAR_IN_OUT 
	r_masterArmCtrlCmd :ST_ArmCtrlCmds;
END_VAR

VAR
	i:INT;
END_VAR
SUPER^.Init(i_masterArm,r_masterArmCtrlCmd);

// disable all joints
m_jntEnableFlag :=g_zeroVec7i;
END_METHOD

END_FUNCTION_BLOCK

// ---- FBs_StateControllers/FB_StateCtrlPerformance.TcPOU
FUNCTION_BLOCK FB_StateCtrlPerformance EXTENDS FB_MasterArmCtrlBase
VAR_INPUT
END_VAR
VAR_OUTPUT
END_VAR
VAR CONSTANT
	//max number of data recording points
	m_dataSum:INT:=8000;
END_VAR

VAR
	//test step
	m_testStep:INT:=-1;
	
	//test joint
	m_testJnt:INT;
	
	//Extreme joint position
	m_minJntPos: ARRAY[1..g_mJntNum] OF LREAL;
	m_maxJntPos: ARRAY[1..g_mJntNum] OF LREAL;
	
	//home position
	m_homeJntPos:ARRAY[1..g_mJntNum] OF LREAL;
	
	//Joint motion speed, acceleration, and jerk
	m_caliMaxjntVel:Vec7d:=[7(3.0*g_deg2rad)];
	m_caliMaxjntAcc:Vec7d:=[7(1.0)];
	m_caliMaxjntJerk:Vec7d:=[7(2.0)];
	
	//arm parameters
	m_armId:INT;
	
	//index
	i,j,id,idx:INT;
	
	//trajectory planner
	m_caliTrajIdx: INT := 1;
	m_jntIdx:INT:=1;
	m_caliMotionSegs :INT :=4;
	m_caliPlanner: ARRAY[1..7,1..g_mJntNum] OF FB_TrajMoveJ;
	m_caliPlannerStart: FB_TrajMoveJ;
	
	//speed test variable
	m_speedMaxTest:BOOL;
	
	//sampling interval
	m_samplingInterval:INT:=80;
	
	//Number of data records
	m_dataRecordNum_2,m_dataRecordNum_3:ARRAY[1..g_mJntNum] OF INT;
			
	//The current values of the second and third trajectories
	m_jntCurrentId2:ARRAY[1..m_dataSum,1..g_mJntNum] OF LREAL;
	m_jntCurrentId3:ARRAY[1..m_dataSum,1..g_mJntNum] OF LREAL;
	
	//friction record value
	m_CoulombFriction,m_ViscousFriction:ARRAY[1..m_dataSum,1..g_mJntNum] OF LREAL;
	
	//friction summation
	m_CoulombFrictionSum,m_ViscousFrictionSum:ARRAY[1..g_mJntNum] OF LREAL;
	
	//friction averange
	m_CoulombFrictionAve,m_ViscousFrictionAve:ARRAY[1..g_mJntNum] OF LREAL;
	
	//friction maxmum value
	m_CoulombFrictionMax,m_ViscousFrictionMax:ARRAY[1..g_mJntNum] OF LREAL;
	
	//Dynamic performance testing time
	m_t:LREAL;
	
	//Dynamic performance testing motion range
	m_motionRange:ARRAY[1..g_mJntNum] OF LREAL:=[0.1,0.1,0.1,0.1,0.1,0.1,0.1];
	
	//Starting point for dynamic performance testing
	m_posOffset:ARRAY[1..g_mJntNum] OF LREAL;
	
	//Number of dynamic performance tests
	m_testNum:INT:=5;
	
	//motion Frequency and angular frequency
	//m_Frequency:LREAL:=3; 	m_w:LREAL;
	m_Frequency:LREAL:=1; 	m_w:LREAL;
	
	//motion Frequency and angular frequency for speed test
	m_FrequencySpeed:LREAL:=0.5; 	m_wSpeed:LREAL;
	
	//motion range for maximum speed test
	//m_motionRangeSpeed:ARRAY[1..g_mJntNum] OF LREAL:=[0.6,0.6,0.6,0.6,0.6,0.6,0.6];
	m_motionRangeSpeed:ARRAY[1..g_mJntNum] OF LREAL:=[0.5,0.5,0.5,0.5,0.5,0.5,0.5];
	
	//joint posotion
	initJntPos,startJntPos,endJntPos :Vec7d;
	
	//Motion amplitude and frequency
	m_motionAmplitude:ARRAY[1..g_mJntNum] OF LREAL;
	m_motionRadiusFre:LREAL;	
	m_Fre:LREAL;
	m_testTime:LREAL;
END_VAR

// override this function in each exact controller
METHOD PROTECTED calcCmdJntPos : BOOL

VAR_IN_OUT CONSTANT
	i_slaveIdx :INT;
	i_shoulderPose :ST_Frame;
	i_masterArm :FB_MasterArm;
	i_slaveStatus :ST_SlaveStatus;
END_VAR

CASE m_testStep OF 
	0: //test the motion range/joint friction/joint gap
		IF m_caliPlanner[m_jntIdx,m_caliTrajIdx].isGene = FALSE THEN
			calcCmdJntPos:=FALSE;
			RETURN;
		END_IF
		
		// traj plan
		calcCmdJntPos :=m_caliPlanner[m_jntIdx,m_caliTrajIdx].evaluate(m_timePeriod, jntPos=> m_cmdJntPos, jntVel=>m_cmdJntVel, jntAcc=> m_cmdJntAcc);
		
		// check if to transit to next segment		
		IF(m_timePeriod > m_caliPlanner[m_jntIdx,m_caliTrajIdx].duration) THEN
			m_caliTrajIdx:=m_caliTrajIdx+1;
			m_timePeriod:=0;
			idx:=0;
			id:=0;
			IF (m_caliTrajIdx>m_caliMotionSegs) THEN
				m_jntIdx:=m_jntIdx+1;
				m_caliTrajIdx:=1;				
			END_IF			
		END_IF
		
		//If all joints have been tested, enter the data processing flow
		IF (m_jntIdx>g_mJntNum) THEN
			m_testStep:=10;
		END_IF
		
		//Record the current value during the testing process
		IF (m_caliTrajIdx=2) THEN
			idx:=idx+1;
			IF (idx>=m_samplingInterval) THEN
				idx:=0;
				id:=id+1;
				m_dataRecordNum_2[m_jntIdx]:=id;
				m_jntCurrentId2[id,m_jntIdx]:=i_masterArm.filtJntCurrent[m_jntIdx]*GVL_ArmJointParameters.g_motorDir[m_armId,m_jntIdx];
			END_IF			
		ELSIF (m_caliTrajIdx=3) THEN
			idx:=idx+1;
			IF (idx>=m_samplingInterval) THEN
				idx:=0;
				id:=id+1;
				m_dataRecordNum_3[m_jntIdx]:=id;
				m_jntCurrentId3[id,m_jntIdx]:=i_masterArm.filtJntCurrent[m_jntIdx]*GVL_ArmJointParameters.g_motorDir[m_armId,m_jntIdx];
			END_IF			
		END_IF
		
	
	10: //Process the data from the above steps
		FOR j:=1 TO g_mJntNum BY 1 DO
			id:=0;
			FOR i:=1 TO m_dataRecordNum_2[j] BY 1 DO 
				idx:=m_dataRecordNum_3[j]-i+1;
				IF (idx>0) THEN
					id:=id+1; //Number of groups for recording data
					m_CoulombFriction[i,j]:=(m_jntCurrentId2[i,j]-m_jntCurrentId3[idx,j])/2;
					m_ViscousFriction[i,j]:=(m_jntCurrentId2[i,j]+m_jntCurrentId3[idx,j])/2;
					
					m_CoulombFrictionSum[j]:=m_CoulombFrictionSum[j]+m_CoulombFriction[i,j];
					m_ViscousFrictionSum[j]:=m_ViscousFrictionSum[j]+m_ViscousFriction[i,j];
					
					IF (m_CoulombFriction[i,j]>m_CoulombFrictionMax[j]) THEN
						m_CoulombFrictionMax[j]:=m_CoulombFriction[i,j];
					END_IF
					
					IF (m_ViscousFriction[i,j]>m_ViscousFrictionMax[j]) THEN
						m_ViscousFrictionMax[j]:=m_ViscousFriction[i,j];
					END_IF				
				END_IF				
			END_FOR			
			//Calculate the mean of frictional force
			m_CoulombFrictionAve[j]:=m_CoulombFrictionSum[j]/id;
			m_ViscousFrictionAve[j]:=m_ViscousFrictionSum[j]/id;			
		END_FOR		
		
		i:=1; m_t:=0;
		m_speedMaxTest:=FALSE;
		m_testStep:=20;
		
		
	20: //m_caliPlannerStart initialization		
		IF (m_speedMaxTest=FALSE) THEN
			m_motionAmplitude:=m_motionRange;
        	m_motionRadiusFre:=m_w;
			m_Fre:=m_Frequency;
		ELSE
			m_motionAmplitude:=m_motionRangeSpeed; 
			m_motionRadiusFre:=m_wSpeed;
			m_Fre:=m_FrequencySpeed;
		END_IF
		
		startJntPos:=i_masterArm.curJntPos; 
		endJntPos:=m_homeJntPos; //m_homeJntPos---m_posOffset
		IF (i=1) THEN
			endJntPos[2]:=-1.657;
			endJntPos[3]:=-0.522;
		END_IF		
		m_caliPlannerStart.init(startJntPos,endJntPos,m_caliMaxjntVel, m_caliMaxJntAcc, m_caliMaxJntJerk);
		m_timePeriod:=0;
		m_testStep:=30;
		
		
	30: //move to the start point
		IF m_caliPlannerStart.isGene = FALSE THEN
			calcCmdJntPos:=FALSE;
			RETURN;
		END_IF
		calcCmdJntPos :=m_caliPlannerStart.evaluate(m_timePeriod, jntPos=> m_cmdJntPos, jntVel=>m_cmdJntVel, jntAcc=> m_cmdJntAcc);			
		IF(m_timePeriod > m_caliPlannerStart.duration) THEN			
			m_timePeriod:=0;			
			m_testStep:=40;
		END_IF
		
		
	40: //Dynamic tracking capability test---3HZ
		m_t:=m_t+g_armCtrlCycleTime;
		sinusoidalMotion(posOffset:= endJntPos[i], amplitude:= m_motionAmplitude[i], t:= m_t, w:= m_motionRadiusFre, pos=> m_cmdJntPos[i], vel=> m_cmdJntVel[i], acc=> m_cmdJntAcc[i]);
		m_testTime:=(m_testNum+0.25)/m_Fre;
		
		IF (m_t>m_testTime) THEN
			m_cmdJntVel[i]:=0; 	m_cmdJntAcc[i]:=0;
			i:=i+1;
			m_t:=0;
			m_testStep:=20;
			IF (i=8) AND (m_speedMaxTest=FALSE) THEN
				i:=1;
				m_speedMaxTest:=TRUE;
				m_testStep:=20;
			ELSIF (i=8) AND (m_speedMaxTest=TRUE) THEN
				i:=1;
				m_testStep:=-1;
				m_isFinished:=TRUE;
			END_IF
		END_IF
	
		
	50: //
		
	
	-1: //
END_CASE
END_METHOD

// override this function in each exact controller
// NOTICE: set joint control mode here, and do some initialization if needed
METHOD PUBLIC init : BOOL
VAR_IN_OUT CONSTANT
	i_masterArm	:FB_MasterArm;
END_VAR
VAR_IN_OUT 
	r_masterArmCtrlCmd :ST_ArmCtrlCmds;
END_VAR
VAR
	//
END_VAR
SUPER^.Init(i_masterArm,r_masterArmCtrlCmd);


//arm id and joint position initial
m_armId:=i_masterArm.armIdx;
initJntPos:=i_masterArm.curJntPos;
startJntPos:=initJntPos;
endJntPos:=initJntPos;


//Assignment of joint position limit values and home position
FOR j:=1 TO g_mJntNum BY 1 DO
	m_minJntPos[j]:=GVL_ArmJointParameters.g_minJntPos[m_armId,j]+20*g_deg2Rad;
	m_maxJntPos[j]:=GVL_ArmJointParameters.g_maxJntPos[m_armId,j]-20*g_deg2Rad;
	m_posOffset[j]:=(m_minJntPos[j]+m_maxJntPos[j])/2;
	m_homeJntPos[j]:=GVL_ArmJointCaliData.g_linkEncCaliJntPos[m_armId,j];
END_FOR


//Joint 7 has a wide range of motion and requires special treatment
m_minJntPos[7]:=50*g_deg2Rad;
m_maxJntPos[7]:=-50*g_deg2Rad;


//step/joint id/ trajectory id
m_testStep:=0;
m_caliTrajIdx :=1;
m_jntIdx:=1;


//Trajectory generator initialization
FOR j:=1 TO g_mJntNum BY 1 DO
	FOR id:=1 TO 4 BY 1 DO
		startJntPos:=endJntPos;
		endJntPos:=m_homeJntPos;
		
		IF (j=1) THEN
			endJntPos[2]:=-1.657;
			endJntPos[3]:=-0.522;
		END_IF
		
		IF (id=1) THEN
			endJntPos[j]:=m_minJntPos[j]; //minimum
		ELSIF (id=2) THEN
			endJntPos[j]:=m_maxJntPos[j]; //maximum
		ELSIF (id=3) THEN
			endJntPos[j]:=m_minJntPos[j]; //minimum
		ELSIF (id=4) THEN
			endJntPos[j]:=m_homeJntPos[j]; //home---m_posOffset
		END_IF
		m_caliPlanner[j,id].init(startJntPos,endJntPos,m_caliMaxjntVel, m_caliMaxJntAcc, m_caliMaxJntJerk);
	END_FOR
END_FOR


//Initialization of calculation results
FOR j:=1 TO g_mJntNum BY 1 DO
	m_CoulombFrictionSum[j]:=0; 	m_CoulombFrictionMax[j]:=0; 	m_CoulombFrictionAve[j]:=0;	
	m_ViscousFrictionSum[j]:=0;	 m_ViscousFrictionMax[j]:=0;	 m_ViscousFrictionAve[j]:=0;
END_FOR


//motion frequency
m_w:=2.0*pi*m_Frequency;
m_wSpeed:=2.0*pi*m_FrequencySpeed;


// update commands to arm
copyCmds(r_masterArmCtrlCmd);
END_METHOD

METHOD sinusoidalMotion : BOOL
VAR_INPUT
	posOffset:LREAL;
	amplitude:LREAL;
	t:LREAL; //time
	w:LREAL; //angular frequency
END_VAR

VAR_OUTPUT
	pos:LREAL;
	vel:LREAL;
	acc:LREAL;
END_VAR

VAR
	
END_VAR

pos:=posOffset+amplitude*SIN(w*t);
vel:=amplitude*w*COS(w*t);
acc:=-amplitude*w*w*SIN(w*t);
END_METHOD

END_FUNCTION_BLOCK

// ---- FBs_StateControllers/FB_EndoscopeController.TcPOU
FUNCTION_BLOCK FB_EndoscopeController
VAR_INPUT
END_VAR
VAR_OUTPUT
END_VAR
VAR
	// steering wheel parameter
	m_wheelRadius:LREAL;
	m_wheelHeight:ARRAY[1..2] OF LREAL;
	m_wheelCenter:ARRAY[1..2] OF Vec3d;
	
	// VF position control parameters
	m_VFPts :ARRAY[1..2] OF Vec3d;
	m_VFDeviation :ARRAY[1..2] OF Vec3d;
	m_lastVFDeviation :ARRAY[1..2] OF Vec3d;
	m_VFVel :ARRAY[1..2] OF Vec3d;
	m_VFVelLpf:ARRAY[1..2,1..3] OF FB_LowPassFilter;
	m_VFKp :LREAL := 200;
	m_VFKd :LREAL := 10;
	m_VFForce :ARRAY[1..2] OF Vec3d;
	
	// oritention control parameter
	m_rotTrackKp : LREAL := 200;
	m_maxTrackVel :LREAL := PI;
	m_jnt4AdjustKp : LREAL :=10;
	m_jnt4MaxVel :LREAL :=pi/3 ;
	m_linearVelLb :LREAL := 0.01;
	m_linearVelUb :LREAL :=0.1;	
	m_cartTrackVel :Vec3d;
	
	// master pose in monitor
		tmpVFPt :ARRAY[1..2] OF Vec3d;
	m_masterPoseInView :ARRAY[1..2] OF ST_Frame;
	
	// flag if the controller has finished all its jobs
	m_isFinished:BOOL:=FALSE;
	
	// controller execute time period
	m_timePeriod :LREAL:=0;
	
	// arm control data
	m_cmdJntPos :ARRAY[1..2] OF VEC7d;
	m_cmdJntVel :ARRAY[1..2] OF VEC7d;
	m_cmdJntAcc :ARRAY[1..2] OF VEC7d;
	m_cmdJntTrq :ARRAY[1..2] OF VEC7d;
	m_jntOPMode :ARRAY[1..2] OF Vec7i;
	m_jntEnableFlag :ARRAY[1..2] OF Vec7i;
	m_cmdCartPose :ARRAY[1..2] OF ST_Frame;
	m_cmdCartTwist :ARRAY[1..2] OF Vec6d;
	
END_VAR

// compute the desired joint position of joint 4-7 for orientation tracking
METHOD PROTECTED calcCmdJntPos : BOOL

VAR_IN_OUT CONSTANT
	i_teleSlaveArmIdx:ARRAY[1..2] OF E_MatchedSlaveArmIdx;
	i_shoulderPose:ARRAY[1..2] OF ST_Frame;
	i_masterArm :ARRAY[1..2] OF FB_MasterArm;
	i_slaveStatus : ST_SlaveStatus;
END_VAR
VAR 
	armIdx:INT;
	i,j : INT;
	
	cmdRotInMonitor :Mat3d;
	invRot:Mat3d;
	
	rotT,rotErr:Mat3d;
	angle : LREAL;
	axis,localAxis :Vec3d;
	oriJaco:Mat34;
	oriJt:Mat43;
	oriJJt:Mat3d;
	oriJJtInv:Mat3d;
	oriJPinv:Mat43;
	cartTrackVel:Vec3d;
	jntTrackVel:Vec4d;
	JpinvJ, nullJ:Mat4d;
	eye4d :Mat4d := g_eye4d;
	redunCtrlVel :Vec4d;
	jnt4TrackVel :LREAL;
	
END_VAR
FOR armIdx:=1 TO 2 DO
	// arm position is compliant
	m_cmdCartPose[armIdx].m_pos:= i_masterArm[armIdx].curCartPose.m_pos;
	FOR i:=1 TO 3 DO 
		m_cmdJntPos[armIdx][i]:=i_masterArm[armIdx].curJntPos[i];
		m_cmdJntVel[armIdx][i]:=i_masterArm[armIdx].curJntVel[i];
	END_FOR
	
	
	// update command oritentation if corresponding slave arm is in SlaveArmState_InstruReady state
	IF i_slaveStatus.m_armState[i_teleSlaveArmIdx[armIdx]] = SlaveArmState_InstruReady THEN
		// command rotation in monitor
		cmdRotInMonitor := i_slaveStatus.m_curArmPose[i_teleSlaveArmIdx[armIdx]].m_rot;
		
		// command rotation in master arm base
		matTranspose(i_shoulderPose[armIdx].m_rot, invRot);
		matMultiply(invRot, cmdRotInMonitor, m_cmdCartPose[armIdx].m_rot);
	END_IF


	// compute cartesian tracking velocity
	matTranspose(i_masterArm[armIdx].simCartPose.m_rot, rotT);
	matMultiply(rotT, m_cmdCartPose[armIdx].m_rot, rotErr);
	rot2AngAxis(rotErr, angle=>angle,axis=>localAxis);
	matMultiVec(i_masterArm[armIdx].simCartPose.m_rot, localAxis, axis);
	vecMultiNum(axis, LIMIT(-m_maxTrackVel, angle*m_rotTrackKp, m_maxTrackVel), cartTrackVel);
	m_cartTrackVel :=cartTrackVel;
	
	// compute pinv of orientation jacobian
	FOR i:=1 TO 3 DO
		FOR j:=1 TO 4 DO
			oriJaco[i,j]:=i_masterArm[armIdx].simJaco[i+3,j+3];
		END_FOR
	END_FOR
	matTranspose(oriJaco, oriJt);
	matMultiply(oriJaco ,oriJt , oriJJt);
	invMat3(oriJJt, oriJJtInv);
	matMultiply(oriJt, oriJJtInv, oriJPinv);
	matMultiVec(oriJpinv, cartTrackVel, jntTrackVel);
	
	// calculate nullspace
	matMultiply(oriJPinv, oriJaco, JpinvJ);
	matSub(eye4d , JpinvJ, nullJ);
	
	// redundant velocity
	jnt4TrackVel:=calcRedunVel(i_masterArm[armIdx]);
	redunCtrlVel[1]:=nullJ[1,1]*jnt4TrackVel;
	redunCtrlVel[2]:=nullJ[2,1]*jnt4TrackVel;
	redunCtrlVel[3]:=nullJ[3,1]*jnt4TrackVel;
	redunCtrlVel[4]:=nullJ[4,1]*jnt4TrackVel;
	
	// update final command joint position and velocity
	FOR i :=1 TO 4 DO 
		m_cmdJntVel[armIdx][i+3]:=jntTrackVel[i]+redunCtrlVel[i];
		m_cmdJntPos[armIdx][i+3]:=m_cmdJntPos[armIdx][i+3]+m_cmdJntVel[armIdx][i+3]*g_armCtrlCycleTime;
	END_FOR

END_FOR
END_METHOD

// compute the desired joint torque of joint 1-3 for intuitive force guiding
METHOD PROTECTED calcCmdJntTrq : BOOL

VAR_IN_OUT CONSTANT
	i_teleSlaveArmIdx:ARRAY[1..2] OF E_MatchedSlaveArmIdx;
	i_shoulderPose:ARRAY[1..2] OF ST_Frame;
	i_masterArm :ARRAY[1..2] OF FB_MasterArm;
	i_slaveStatus : ST_SlaveStatus;
END_VAR

VAR 
	
	armIdx :INT;
	i,j :INT;
	kpForce, kdForce :Vec3d;
	jntTrq :Vec3d;
	posJaco, posJacoT :Mat3d;
END_VAR
m_cmdJntTrq[1] := g_zeroVec7d;
m_cmdJntTrq[2] := g_zeroVec7d;

// compute cuurent VF parameters
steeringWheelCalc(i_shoulderPose, i_masterArm);

// compute VF motion velocity
FOR armIdx:=1 TO 2 DO
	vecSub(m_lastVFDeviation[armIdx],m_VFDeviation[armIdx], m_VFVel[armIdx]);
	vecSelfMultiNum(m_VFVel[armIdx], g_armCtrlFreq);
	FOR j:=1 TO 3 DO 
		m_VFVel[armIdx][j] := m_VFVelLpf[armIdx,j].run(m_VFVel[armIdx][j]);
	END_FOR
	
	m_lastVFDeviation[armIdx] := m_VFDeviation[armIdx];
END_FOR

// compute VF force
FOR armIdx:=1 TO 2 DO
	vecMultiNum(m_VFDeviation[armIdx], m_VFKp, kpForce);
	vecMultiNum(m_VFVel[armIdx], m_VFKd, kdForce);
	vecSub(kpForce, kdForce, m_VFForce[armIdx]);
END_FOR

// compute joint space torque
FOR armIdx:=1 TO 2 DO 
	FOR i :=1 TO  3 DO
		FOR j:=1 TO 3 DO
			posJaco[i,j]:= i_masterArm[armIdx].jaco[i,j];
		END_FOR
	END_FOR
	matTranspose(posJaco, posJacoT);
	matMultiVec(posJacoT, m_VFForce[armIdx], jntTrq);
	
	m_cmdJntTrq[armIdx][1]:=jntTrq[1];
	m_cmdJntTrq[armIdx][2]:=jntTrq[2];
	m_cmdJntTrq[armIdx][3]:=jntTrq[3];
END_FOR
END_METHOD

METHOD PROTECTED calcRedunVel : LREAL
VAR_IN_OUT CONSTANT
	i_masterArm :FB_MasterArm;
END_VAR

VAR 
	j6Bias,j5Bias :LREAL;
	velScale :LREAL;
	linearVel :Vec3d;
	curJntPos : Vec7d;
	jnt4LinkPos :LREAL;
END_VAR
// compute desired joint4 link position
curJntPos :=  i_masterArm.cmdJntPos;
jnt4LinkPos:=i_masterArm.jnt4MotorToLink(curJntPos[2],curJntPos[3],curJntPos[4]);
IF 1= i_masterArm.armIdx THEN
	j6Bias :=curJntPos[6]+PI/2;
ELSE 
	j6Bias := curJntPos[6]-PI/2;
END_IF

// scale based on joint5 position
j5Bias :=  LIMIT (0, ABS(curJntPos[5] -pi), pi/2);
j6Bias := j6Bias * ABS(COS(j5Bias));

// scale based on linear velocity
linearVel[1]:=i_masterArm.curCartTwist[1];
linearVel[2]:=i_masterArm.curCartTwist[2];
linearVel[3]:=i_masterArm.curCartTwist[3];
velScale :=LIMIT(0, (norm(linearVel)-m_linearVelLb)/(m_linearVelUb-m_linearVelLb),1.0);


calcRedunVel := LIMIT(-m_jnt4MaxVel, -j6Bias * m_jnt4AdjustKp * velScale ,m_jnt4MaxVel);

// joint limit
IF (calcRedunVel > 0 AND jnt4LinkPos+calcRedunVel * g_armCtrlCycleTime > GVL_ArmJointParameters.g_maxJntPos[i_masterArm.armIdx,4])
	 OR ( calcRedunVel <0 AND  jnt4LinkPos +calcRedunVel * g_armCtrlCycleTime< GVL_ArmJointParameters.g_minJntPos[i_masterArm.armIdx,4]) THEN
	 calcRedunVel :=0;
END_IF
END_METHOD

// override this function in each exact controller
// NOTICE: set joint control mode here, and do some initialization if needed
METHOD PUBLIC init : BOOL
VAR_IN_OUT CONSTANT
	i_shoulderPose:ARRAY[1..2] OF ST_Frame;
	i_masterArm :ARRAY[1..2] OF FB_MasterArm;
END_VAR
VAR_IN_OUT 
	r_masterArmCtrlCmd :ARRAY[1..2] OF ST_ArmCtrlCmds;
END_VAR
VAR
	i,j:INT;
END_VAR
m_timePeriod:=0;
FOR i:=1 TO 2 DO 
	m_jntEnableFlag[i] :=g_onesVec7i;
	m_jntOPMode[i][1] := DriverOPMode_Trq;
	m_jntOPMode[i][2] := DriverOPMode_Trq;
	m_jntOPMode[i][3] := DriverOPMode_Trq;
	m_jntOPMode[i][4] := DriverOPMode_PosTrq;
	m_jntOPMode[i][5] := DriverOPMode_PosTrq;
	m_jntOPMode[i][6] := DriverOPMode_PosTrq;
	m_jntOPMode[i][7] := DriverOPMode_PosTrq;
	m_cmdCartPose[i]:=i_masterArm[i].curCartPose;
	m_cmdCartTwist[i]:=g_zeroVec6d;
	m_cmdJntPos[i]:=i_masterArm[i].curJntPos;
	m_cmdJntVel[i]:=g_zeroVec7d;
	m_cmdJntAcc[i]:=g_zeroVec7d;
	m_cmdJntTrq[i]:=g_zeroVec7d;
	
	r_masterArmCtrlCmd[i].m_jntEnableFlag :=m_jntEnableFlag[i];
	r_masterArmCtrlCmd[i].m_cmdCartPose:=m_cmdCartPose[i];
	r_masterArmCtrlCmd[i].m_cmdCartTwist:=m_cmdCartTwist[i];
	r_masterArmCtrlCmd[i].m_cmdJntPos:=m_cmdJntPos[i];
	r_masterArmCtrlCmd[i].m_cmdJntVel:=m_cmdJntVel[i];
	r_masterArmCtrlCmd[i].m_cmdJntAcc:=m_cmdJntAcc[i];
	r_masterArmCtrlCmd[i].m_cmdJntTrq:=m_cmdJntTrq[i];
	r_masterArmCtrlCmd[i].m_jntOPMode:=m_jntOPMode[i];
	
	m_lastVFDeviation[i] := g_zeroVec3d;
	
	// filter init
	FOR j:=1 TO 3 DO 
		m_VFVelLpf[i,j].init(1, g_curJntVelLpfCutoffFreq, g_armCtrlFreq);
	END_FOR

END_FOR

steeringWheelInit(i_shoulderPose, i_masterArm);
END_METHOD

// TODO: corner case that two arm tips coincide on z axis need to be handle
METHOD run : BOOL

VAR_IN_OUT CONSTANT
	i_teleSlaveArmIdx:ARRAY[1..2] OF E_MatchedSlaveArmIdx;
	i_shoulderPose:ARRAY[1..2] OF ST_Frame;
	i_masterArm :ARRAY[1..2] OF FB_MasterArm;
	i_slaveStatus : ST_SlaveStatus;
END_VAR
VAR_IN_OUT 
	r_masterArmCtrlCmd :ARRAY[1..2] OF ST_ArmCtrlCmds;
END_VAR
VAR
	i:INT;
END_VAR
IF m_isFinished THEN
	RETURN;
END_IF

// check if arm enabled
IF NOT(i_masterArm[1].isEnabled(m_jntEnableFlag[1])) OR NOT(i_masterArm[2].isEnabled(m_jntEnableFlag[2]))  THEN
	RETURN;
END_IF

// calculate command joint position--Motion control
calcCmdJntPos(i_teleSlaveArmIdx, i_shoulderPose, i_masterArm,i_slaveStatus);

// calculate command joint torque -- Force control
calcCmdJntTrq(i_teleSlaveArmIdx, i_shoulderPose, i_masterArm,i_slaveStatus);

// update commands to arm
FOR i:=1 TO 2 DO 
	r_masterArmCtrlCmd[i].m_cmdJntPos:=m_cmdJntPos[i];
	r_masterArmCtrlCmd[i].m_cmdJntTrq:=m_cmdJntTrq[i];
END_FOR

// update time period
m_timePeriod := m_timePeriod+g_armCtrlCycleTime;
END_METHOD

METHOD PROTECTED steeringWheelCalc : BOOL
VAR_IN_OUT CONSTANT
	i_shoulderPose:ARRAY[1..2] OF ST_Frame;
	i_masterArm :ARRAY[1..2] OF FB_MasterArm;
END_VAR
VAR
	tipCenter :Vec3d;
	i:INT;

	rotT :Mat3d;
	VFDeviationInView:Vec3d;
END_VAR
// master pose in view coordinate
m_masterPoseInView[1] := transform(i_shoulderPose[1],  i_masterArm[1].curCartPose);
m_masterPoseInView[2] := transform(i_shoulderPose[2],  i_masterArm[2].curCartPose);

// master tip center 
vecAdd(m_masterPoseInView[1].m_pos, m_masterPoseInView[2].m_pos, tipCenter);
vecSelfMultiNum(tipCenter,0.5);

FOR i:=1 TO 2 DO 
	// steering wheel center 
	m_wheelCenter[i]:=tipCenter;
	m_wheelCenter[i][3]:=m_wheelCenter[i][3]+m_wheelHeight[i];
	
	// compute current virtual fixture points on wheel 
	vecSub(m_masterPoseInView[i].m_pos, m_wheelCenter[i], tmpVFPt[i]);
	tmpVFPt[i][3]:=0;
	IF NOT(normalize(tmpVFPt[i])) THEN
		steeringWheelCalc := FALSE;
		RETURN;
	END_IF
	vecSelfMultiNum(tmpVFPt[i], m_wheelRadius);
	vecAdd(m_wheelCenter[i], tmpVFPt[i], m_VFPts[i]);
	
	// compute current deviation from VF points in shoulder coordinate
	vecSub(m_VFPts[i], m_masterPoseInView[i].m_pos, VFDeviationInView);
	matTranspose(i_shoulderPose[i].m_rot , rotT);
	matMultiVec(rotT, VFDeviationInView, m_VFDeviation[i]);

END_FOR
END_METHOD

METHOD PROTECTED steeringWheelInit : BOOL
VAR_IN_OUT CONSTANT
	i_shoulderPose:ARRAY[1..2] OF ST_Frame;
	i_masterArm :ARRAY[1..2] OF FB_MasterArm;
END_VAR
VAR
	tipDis,tipCenter :Vec3d;
END_VAR
// master pose in view coordinate
m_masterPoseInView[1] := transform(i_shoulderPose[1],  i_masterArm[1].curCartPose);
m_masterPoseInView[2] := transform(i_shoulderPose[2],  i_masterArm[2].curCartPose);

// master tip height relative to center 
vecAdd(m_masterPoseInView[1].m_pos, m_masterPoseInView[2].m_pos, tipCenter);
vecSelfMultiNum(tipCenter,0.5);
m_wheelHeight[1] :=m_masterPoseInView[1].m_pos[3] -  tipCenter[3];
m_wheelHeight[2] :=m_masterPoseInView[2].m_pos[3] -  tipCenter[3];

// master tip distance  relative to center 
vecSub(m_masterPoseInView[1].m_pos, m_masterPoseInView[2].m_pos, tipDis);
tipDis[3] := 0;
m_wheelRadius :=norm(tipDis)/2.0;
END_METHOD

END_FUNCTION_BLOCK

// ---- AgiMaths/Frames/rotY.TcPOU
FUNCTION rotY : mat3d
VAR_INPUT
	i_ang : LREAL;
END_VAR
VAR
	rot :Mat3d := g_eye3d;
END_VAR

rot[1,1]:=COS(i_ang);
rot[3,3]:=rot[1,1];
rot[1,3]:=SIN(i_ang);
rot[3,1]:=-rot[1,3];
rotY:=rot;

END_FUNCTION

// ---- Mains/RobotDynamics.TcPOU
PROGRAM RobotDynamics

VAR
	// master robot arms joint data
	m_masterJointsData AT %I* :ST_MasterJointData;
	
	// dynamic output
	m_masterDynaData AT %Q* : ST_MasterDynaData;
	
	// flag to init robot dynamic model
	m_robotDynaInit :BOOL :=FALSE;
	
	// master grivity model 
	m_gravityModel :ARRAY[1..g_mArmNum] OF FB_MasterGravity;
	
	// master arm dynamic model
	m_armDynamic :ARRAY[1..g_mArmNum] OF FB_MasterDynamic;
	
	// master friction model
	m_frictionModel : ARRAY[1..g_mArmNum] OF FB_MasterFriciton;
	
	// master external torque observer
	m_jntDOB : ARRAY[1..g_mArmNum] OF FB_JntObserver;
	
	// code execute time measure
	m_codeTime : Profiler;
	
	i: INT;
	
END_VAR

m_codeTime(START:=TRUE, RESET:=TRUE);

// robot dynamic model init
IF m_robotDynaInit =FALSE THEN
	FOR i:=1 TO g_mArmNum DO
		m_gravityModel[i].Init(i);
		m_armDynamic[i].init(i);
		m_frictionModel[i].init(i);
		// NOTE: curJntPos is usually zero when init, so observer need some time to stable after code run
		m_jntDOB[i].init(i, m_masterJointsData.m_curJntPos[i]); 
	END_FOR

	m_robotDynaInit:=TRUE;
END_IF

FOR i:=1 TO g_mArmNum DO
	// run gravity model
	m_gravityModel[i].run(m_masterJointsData.m_curLinkPos[i], m_masterDynaData.m_gravity[i]);
	
	// run dynamic model
	m_armDynamic[i].updateDynamic(m_masterJointsData.m_curJntPos[i]);
	m_masterDynaData.m_massMat[i]:=m_armDynamic[i].jntMassMat;
	m_masterDynaData.m_lambda[i]:=m_armDynamic[i].cartMassMat;
	m_masterDynaData.m_dynaNullspace[i]:=m_armDynamic[i].dynaNullspace;
	
	// run friction model
	m_masterDynaData.m_friction[i] := m_frictionModel[i].run(m_masterDynaData.m_gravity[i],m_masterJointsData.m_curJntVel[i]);
	
(*	// run DOB
	 m_masterDynaData.m_jntExtTrq[i] := m_jntDOB[i].run(m_masterJointsData.m_curJntTrq[i], m_masterJointsData.m_curJntPos[i], m_masterDynaData.m_massMat[i]);
	// remove gravity and friction from external torque
	vecSelfAdd(m_masterDynaData.m_jntExtTrq[i], m_masterDynaData.m_gravity[i]);
	vecSelfAdd(m_masterDynaData.m_jntExtTrq[i], m_masterDynaData.m_friction[i]);*)
	
END_FOR

m_codeTime(START:=FALSE);

END_PROGRAM

// ---- FBs_RobotDynamics/FB_MasterGravity.TcPOU
FUNCTION_BLOCK FB_MasterGravity
VAR_INPUT
END_VAR
VAR_OUTPUT
END_VAR
VAR
	// arm index
	m_armIdx :INT;
	
	(*graParam=[ 2.7244*m3 + 2.7244*m4 + 2.7244*m5 + 2.7244*m6 + 9.8*mx2 + 9.8*mx9,
            	9.8*my2 + 9.8*my9,
			 	3.577*m4 + 3.577*m5 + 3.577*m6 + 0.49*m9 + 9.8*mx3 + 9.8*mx8
           		1.5827*m4 + 1.5827*m5 + 1.5827*m6 + 9.8*my3 + 9.8*my8 + 9.8*mz4
            	mz5-my4,	my5+mz6,  	mx4,   	mx5, 	mx6,   	my6
            	preF2,   k2,   preF3,    k3,    preF5   k5]*)
	m_gravityParam :ARRAY[1..16] OF REAL;
	// spring2 [L0, b1, b2, l1, r0]
	m_spring2Param :ARRAY[1..5] OF LREAL;
	// spring3 [L0, b1, b2, l1, r0,d]
	m_spring3Param :ARRAY[1..6] OF LREAL;
	// spring5 [L0, s1, L1, r0, beta]
	m_spring5Param :ARRAY[1..5] OF LREAL;
	
	// gravity deviation
	m_gravityDeviation :Vec7d;
END_VAR

METHOD protected getRegMat : BOOL
VAR_INPUT
	// 0 for left, 1 for right
	i_armIdx:INT;
END_VAR
VAR_IN_OUT CONSTANT
	// position of all the active joint
	i_jointPos:ARRAY[1..7] OF LREAL;
END_VAR
VAR_IN_OUT
	o_regMat:ARRAY[1..5,1..16] OF LREAL;
END_VAR
VAR
	q2,q8,q4,q5,q6:LREAL;
	i,j :INT;
END_VAR
q2:=i_jointPos[2];
q8:=i_jointPos[3];
q4:=i_jointPos[4];
q5:=i_jointPos[5];
q6:=i_jointPos[6];

FOR i:=1 TO 5 DO
	FOR j:=1 TO 16 DO
		o_regMat[i,j]:=0;
	END_FOR
END_FOR

// active joint 2
o_regMat[1,1]:=COS(q2);
o_regMat[1,2]:=-SIN(q2); 
o_regMat[1,3] := 0;
o_regMat[1,4] :=   0;
o_regMat[1,5] := - 4.9*(COS(q2 - q4) - COS(q4 - q2 + 2.0*q8));
o_regMat[1,6] :=  9.8*COS(q4 - q2 + q8)*SIN(q5)*SIN(q8);
o_regMat[1,7] :=   - 4.9*(SIN(q2 - q4) + SIN(q4 - q2 + 2.0*q8));
o_regMat[1,8] :=   - 9.8*COS(q4 - q2 + q8)*COS(q5)*SIN(q8);
o_regMat[1,9] :=  9.8*SIN(q8)*(SIN(q4 - q2 + q8)*SIN(q6) - COS(q4 - q2 + q8)*COS(q5)*COS(q6));
o_regMat[1,10] :=9.8*SIN(q8)*(SIN(q4 - q2 + q8)*COS(q6) + COS(q4 - q2 + q8)*COS(q5)*SIN(q6));
spring2RegMat(q2, o_preF=>o_regMat[1,11], o_stiff=>o_regMat[1,12]);
o_regMat[1,11]:=-o_regMat[1,11];         
o_regMat[1,12]:=-o_regMat[1,12];

// active joint3
o_regMat[2,3]:= COS(q8);
o_regMat[2,4]:= - SIN(q8);
o_regMat[2,5]:= -9.8*(COS(2.0*q8)*COS(q2)*COS(q4) + COS(2.0*q8)*SIN(q2)*SIN(q4) - SIN(2.0*q8)*COS(q2)*SIN(q4) + SIN(2.0*q8)*COS(q4)*SIN(q2));
o_regMat[2,6]:= -9.8*(COS(q5)*SIN(q8) + COS(2.0*q8)*COS(q2)*SIN(q4)*SIN(q5) - COS(2.0*q8)*COS(q4)*SIN(q2)*SIN(q5) + SIN(2.0*q8)*COS(q2)*COS(q4)*SIN(q5) + SIN(2.0*q8)*SIN(q2)*SIN(q4)*SIN(q5));
o_regMat[2,7]:= 9.8*(COS(2.0*q8)*COS(q2)*SIN(q4) - COS(2.0*q8)*COS(q4)*SIN(q2) + SIN(2.0*q8)*COS(q2)*COS(q4) + SIN(2.0*q8)*SIN(q2)*SIN(q4));
o_regMat[2,8]:= 9.8*(COS(2.0*q8)*COS(q2)*COS(q5)*SIN(q4) - SIN(q5)*SIN(q8) - COS(2.0*q8)*COS(q4)*COS(q5)*SIN(q2) + SIN(2.0*q8)*COS(q2)*COS(q4)*COS(q5) + SIN(2.0*q8)*COS(q5)*SIN(q2)*SIN(q4));
o_regMat[2,9]:= 9.8*(COS(2.0*q8)*COS(q2)*COS(q4)*SIN(q6) - COS(q6)*SIN(q5)*SIN(q8) + COS(2.0*q8)*SIN(q2)*SIN(q4)*SIN(q6) - SIN(2.0*q8)*COS(q2)*SIN(q4)*SIN(q6) + SIN(2.0*q8)*COS(q4)*SIN(q2)*SIN(q6) + COS(2.0*q8)*COS(q2)*COS(q5)*COS(q6)*SIN(q4) - COS(2.0*q8)*COS(q4)*COS(q5)*COS(q6)*SIN(q2) + SIN(2.0*q8)*COS(q2)*COS(q4)*COS(q5)*COS(q6) + SIN(2.0*q8)*COS(q5)*COS(q6)*SIN(q2)*SIN(q4)); 
o_regMat[2,10]:= 9.8*(SIN(q5)*SIN(q6)*SIN(q8) + COS(2.0*q8)*COS(q2)*COS(q4)*COS(q6) + COS(2.0*q8)*COS(q6)*SIN(q2)*SIN(q4) - SIN(2.0*q8)*COS(q2)*COS(q6)*SIN(q4) + SIN(2.0*q8)*COS(q4)*COS(q6)*SIN(q2) - COS(2.0*q8)*COS(q2)*COS(q5)*SIN(q4)*SIN(q6) + COS(2.0*q8)*COS(q4)*COS(q5)*SIN(q2)*SIN(q6) - SIN(2.0*q8)*COS(q2)*COS(q4)*COS(q5)*SIN(q6) - SIN(2.0*q8)*COS(q5)*SIN(q2)*SIN(q4)*SIN(q6));
spring3RegMat(q8, o_preF=>o_regMat[2,13], o_stiff=>o_regMat[2,14]);
o_regMat[2,13]:=-o_regMat[2,13];
o_regMat[2,14]:=-o_regMat[2,14];

// active joint4
o_regMat[3,5]:= 9.8*SIN(q4 - q2 + q8)*SIN(q8);
o_regMat[3,6]:= - 9.8*COS(q4 - q2 + q8)*SIN(q5)*SIN(q8);
o_regMat[3,7]:= 9.8*COS(q4 - q2 + q8)*SIN(q8);
o_regMat[3,8]:= 9.8*COS(q4 - q2 + q8)*COS(q5)*SIN(q8);
o_regMat[3,9]:= - 9.8 *SIN(q8)*(SIN(q4 - q2 + q8)*SIN(q6) - COS(q4 - q2 + q8)*COS(q5)*COS(q6));
o_regMat[3,10]:= - 9.8*SIN(q8)*(SIN(q4 - q2 + q8)*COS(q6) + COS(q4 - q2 + q8)*COS(q5)*SIN(q6));
              
// active joint5
o_regMat[4,6]:= -9.8* (COS(q8)*SIN(q5) + SIN(q4 - q2 + q8)*COS(q5)*SIN(q8));
o_regMat[4,7]:= 0;
o_regMat[4,8]:= 9.8* (COS(q5)*COS(q8) - SIN(q4 - q2 + q8)*SIN(q5)*SIN(q8));
o_regMat[4,9]:= 9.8*COS(q6)*(COS(q5)*COS(q8) - SIN(q4 - q2 + q8)*SIN(q5)*SIN(q8));
o_regMat[4,10]:= -9.8*SIN(q6)*(COS(q5)*COS(q8) - SIN(q4 - q2 + q8)*SIN(q5)*SIN(q8));
spring5RegMat(q5, o_preF=>o_regMat[4,15], o_stiff=>o_regMat[4,16]);
o_regMat[4,15]:=-o_regMat[4,15];
o_regMat[4,16]:=-o_regMat[4,16];

// active joint5
o_regMat[5,9]:= -9.8*(COS(q8)*SIN(q5)*SIN(q6) - COS(q4 - q2 + q8)*COS(q6)*SIN(q8) + SIN(q4 - q2 + q8)*COS(q5)*SIN(q6)*SIN(q8));
o_regMat[5,10]:= -9.8*(COS(q4 - q2 + q8)*SIN(q6)*SIN(q8) + COS(q6)*COS(q8)*SIN(q5) + SIN(q4 - q2 + q8)*COS(q5)*COS(q6)*SIN(q8));
END_METHOD

METHOD PUBLIC init : BOOL
VAR_INPUT
	i_armIdx :INT;
END_VAR
VAR
	i:INT;
END_VAR
m_armIdx:=i_armIdx;

FOR i:=1 TO 16 DO
	m_gravityParam[i]:=GVL_ArmDynamics.g_gravityParam[m_armIdx, i];
END_FOR

FOR i:=1 TO 5 DO
	m_spring2Param[i]:=GVL_ArmDynamics.g_spring2Param[i];
	m_spring3Param[i]:=GVL_ArmDynamics.g_spring3Param[i];
	m_spring5Param[i]:=GVL_ArmDynamics.g_spring5Param[i];
END_FOR
m_spring3Param[6]:=GVL_ArmDynamics.g_spring3Param[6];

FOR i:=1 TO 7 DO
	m_gravityDeviation[i]:=GVL_ArmDynamics.g_gravityDeviaion[m_armIdx, i];
END_FOR
END_METHOD

METHOD PUBLIC run : BOOL
VAR_IN_OUT CONSTANT
	// active joint position
	i_jntPos :vec7d;
END_VAR
VAR_IN_OUT
	r_gravity :Vec7d;
END_VAR
VAR
	// gravity regression matrix
	regMat:ARRAY[1..5,1..16] OF LREAL;
	
	i,j:INT;
END_VAR
getRegMat(m_armIdx,i_jntPos,regMat);

FOR i:=2 TO 6 DO
	r_gravity[i]:=0;
	FOR j:=1 TO 16 DO
		r_gravity[i]:=r_gravity[i]+regMat[i-1,j]*m_gravityParam[j];
	END_FOR
	
	// add bias torque
	r_gravity[i]:= r_gravity[i] + m_gravityDeviation[i];
END_FOR
END_METHOD

(*spring force F = preF+k(L-L0)
% torque trq=F*t=preF*t+k*t*(L-L0)=[t, t*(L-L0)]*[preF,k]'
% this function return [t, t(L-L0)]*)
METHOD PROTECTED spring2RegMat : BOOL
VAR_INPUT
	i_q2:LREAL;
END_VAR

VAR
	// spring paramters
	L0, b1, b2, l1, r0 : LREAL;

	theta,length,t:LREAL;  
	
END_VAR

VAR_OUTPUT
	o_preF:LREAL;
	o_stiff:LREAL;
END_VAR
L0:=m_spring2Param[1]; 
b1:=m_spring2Param[2]; 
b2:=m_spring2Param[3]; 
l1:=m_spring2Param[4]; 
r0:=m_spring2Param[5]; 

L0:=L0+b1+b2;
 
//spring length
theta:=i_q2+90*g_deg2Rad;
length:=SQRT(l1*l1+r0*r0+2*l1*r0*COS(theta));

//force arm
t:=r0*l1*SIN(theta)/Length;

//torque direction is determined by theta(or t)
o_preF:=t;
o_stiff:=t*(length-L0);
END_METHOD

(*spring force F = preF+k(L-L0)
% torque trq=F*t=preF*t+k*t*(L-L0)=[t, t*(L-L0)]*[preF,k]'
% this function return [t, t(L-L0)]*)
METHOD PROTECTED spring3RegMat : BOOL
VAR_INPUT
	i_q3:LREAL;
END_VAR

VAR
	// spring paramters
	L0, b1, b2, l1, r0, d: LREAL;

	alpha, beta,tanBeta, length,t:LREAL;  
	
	spring: INT;
END_VAR

VAR_OUTPUT
	o_preF:LREAL;
	o_stiff:LREAL;
END_VAR
L0:=m_spring3Param[1]; 
b1:=m_spring3Param[2]; 
b2:=m_spring3Param[3]; 
l1:=m_spring3Param[4]; 
r0:=m_spring3Param[5];
d:=m_spring3Param[6];

L0:=L0+b1+b2;
 
// spring length
    alpha:=i_q3+90*g_deg2Rad;
    tanBeta:=(r0*SIN(alpha)+d)/(l1+r0*COS(alpha));
    beta:=ATAN(tanBeta);
    length:=d/SIN(beta)+r0*SIN(alpha)/SIN(beta);
    
// force arm
    t:=(l1-d*cot(beta))*SIN(beta);
    
// torque direction is determined by theta(or t)
    o_preF:=t;
    o_stiff:=t*(length-L0);
END_METHOD

(*spring force F = preF+k(L-L0)
 torque trq=F*t=preF*t+k*t*(L-L0)=[t, t*(L-L0)]*[preF,k]'
 this function return [t, t(L-L0)]
 armIdx, 0 for left arm , 1 for right arm]*)
METHOD PROTECTED spring5RegMat : BOOL
VAR_INPUT
	i_q5:LREAL;
END_VAR

VAR
	// spring paramters
	L0, s1, L1, r0, beta: LREAL;

	theta, length,t:LREAL;  
	
	spring: INT;
	joint: INT;
	armIdx: INT;
	b1: LREAL;
END_VAR

VAR_OUTPUT
	o_preF:LREAL;
	o_stiff:LREAL;
END_VAR
L0:=m_spring5Param[1]; 
s1:=m_spring5Param[2]; 
L1:=m_spring5Param[3]; 
r0:=m_spring5Param[4]; 
beta:=m_spring5Param[5];

L0:=L0+s1;
 
// joint 5 motion angle
IF 1=m_armIdx THEN 
	theta:=i_q5-pi;// left arm
ELSE
	theta:=pi-i_q5; // right arm
END_IF

// spring length and force arm
length:=SQRT(L1*L1+r0*r0+2*L1*r0*COS(theta+beta));
t:=L1*r0*SIN(theta+beta)/length;

// torque direction is determined by t
IF 1=m_armIdx THEN 
	o_preF:=t;
	o_stiff:=t*(length-L0);
else
	o_preF:=-t;
	o_stiff:=-t*(length-L0);
END_IF
END_METHOD

END_FUNCTION_BLOCK

// ---- FBs_RobotDynamics/FB_MasterDynamic.TcPOU
FUNCTION_BLOCK FB_MasterDynamic
VAR_INPUT
END_VAR
VAR_OUTPUT
END_VAR
VAR
	m_armIdx :INT;
	//kinematic constraint
	//  q3 = q8 - q2;            qdot3=qdot8-qdot2;
	//  q9 = q2-q8;              qdot9=qdot2-qdot8;
	//  q4= q4motor+q8-q2-90;    qdot4=qdot4m+qdot8
 	// jacobian with active joints
 	// jaco_DH*qdot_DH = jaco_DH * (A * qdot_active)= jaco * qdot_active
 	// q_DH=[q1,q2,q3,q4,q5,q6,q7,q8,q9];
 	// q_active=[q1,q2,q8,q4m,q5,q6,q7]
	m_jacoA :ARRAY[1..9,1..7] OF LREAL:=
		[   1,  0,  0,  0,  0,  0,  0,
			0,  1,  0,  0,  0,  0,  0,
			0, -1,  1,  0,  0,  0,  0,
			0, -1,  1,  1,  0,  0,  0,
			0,  0,  0,  0,  1,  0,  0,
			0,  0,  0,  0,  0,  1,  0,
			0,  0,  0,  0,  0,  0,  1,
			0,  0,  1,  0,  0,  0,  0,
			0,  1, -1,  0,  0,  0,  0];
	
	// DH parameters
	m_armDH:ARRAY[1..9] OF Vec4d;// last column is joint position
	m_d1, m_a3,m_a4,m_d4,m_a9 :LREAL;
	
	// dynamic parameters
	m_linkMass :ARRAY[1..9] OF LREAL;
	m_linkCOM :ARRAY[1..9] OF Vec3d;
	m_linkInertia :ARRAY[1..9] OF Mat3d;
		
	// frame of each joint
	m_jntFrame :ARRAY[1..9] OF ST_Frame;
	
	// jacobian of mass center
	m_Jp :ARRAY[1..9] OF Mat37;
	m_Jo :ARRAY[1..9] OF Mat37;
	
	// tcp jacobian
	m_jaco : Mat67;
	
	// motor inertia at link size
	m_motorInertia :Vec7d;
	
	// mass matrix in joint space
	m_massMat :Mat7d;
	m_massMatInv:Mat7d;
	
	// mass matrix in cartesian space
	m_lambdaInv :Mat6d;
	m_lambda :Mat6d;
	
	// dynamic nullspace(I-J'*inv(J'))
	m_JtGeneInv :Mat67;
	m_dynaNullspace : Mat7d;
	
END_VAR

PROPERTY PUBLIC cartMassMat : Mat6d
GET
cartMassMat := m_lambda;
END_GET
END_PROPERTY

PROPERTY PUBLIC dynaNullspace : Mat7d
GET
dynaNullspace:=m_dynaNullspace;
END_GET
END_PROPERTY

METHOD init : BOOL
VAR_INPUT
	i_armIdx :INT ;
END_VAR

VAR
	i:INT;
END_VAR
m_armIdx:=i_armIdx;
m_d1:=g_d1;
m_a3:=g_a3;
m_a4:=g_a4;
m_d4:=g_d4;
m_a9:=g_a9;

m_linkMass:=GVL_ArmDynamics.g_linkMass;
FOR i:=1 TO 9 DO
	m_linkCOM[i][1]:=GVL_ArmDynamics.g_linkCOM[i,1];
	m_linkCOM[i][2]:=GVL_ArmDynamics.g_linkCOM[i,2];
	m_linkCOM[i][3]:=GVL_ArmDynamics.g_linkCOM[i,3];
	
	m_armDH[i][1]:=g_masterArmDH[i,1];
	m_armDH[i][2]:=g_masterArmDH[i,2];
	m_armDH[i][3]:=g_masterArmDH[i,3];
	m_armDH[i][4]:=g_masterArmDH[i,4];
	
	m_linkInertia[i][1,1]:=GVL_ArmDynamics.g_linkInertia[i,1];
	m_linkInertia[i][2,2]:=GVL_ArmDynamics.g_linkInertia[i,2];
	m_linkInertia[i][3,3]:=GVL_ArmDynamics.g_linkInertia[i,3];
	m_linkInertia[i][1,2]:=GVL_ArmDynamics.g_linkInertia[i,4];
	m_linkInertia[i][1,3]:=GVL_ArmDynamics.g_linkInertia[i,5];
	m_linkInertia[i][2,3]:=GVL_ArmDynamics.g_linkInertia[i,6];
	m_linkInertia[i][2,1]:=m_linkInertia[i][1,2];
	m_linkInertia[i][3,1]:=m_linkInertia[i][1,3];
	m_linkInertia[i][3,2]:=m_linkInertia[i][2,3];
END_FOR

FOR i:=1 TO 7 DO
	m_motorInertia[i]:=GVL_ArmDynamics.g_motorInertia[i]*GVL_ArmJointParameters.g_motorReduction[i]*GVL_ArmJointParameters.g_motorReduction[i];
END_FOR
END_METHOD

PROPERTY PUBLIC jntMassMat : Mat7d
GET
jntMassMat := m_massMat;
END_GET
END_PROPERTY

// update dynamic and kinematic data 
METHOD updateDynamic : BOOL
VAR_IN_OUT CONSTANT
	i_jntPos : Vec7d;
END_VAR
VAR
	
	i,j:INT;
	m,n :INT;
	linkMassMat :ARRAY[1..9] OF Mat7d;
	linkInerMat :ARRAY[1..9] OF Mat7d;
	inertia,Rt :Mat3d;
	JotI :ARRAY[1..7,1..3] OF LREAL;
	Jot :ARRAY[1..7,1..3] OF LREAL;
	Jpt :ARRAY[1..7,1..3] OF LREAL;
	
	tmpMat3d :Mat3d;
	tmpMat67: Mat67;
	tmpMat7d : Mat7d;
	jacoT: Mat76;
	
END_VAR
// update kinematic 
updateKinematic(i_jntPos);

// joint space mass matrix
// massMat=m*Jp'*Jp+Jo'*R*I*R'*Jo
FOR i:=1 TO 9 DO
	// iner=R*I*R'
	matMultiply(m_jntFrame[i].m_rot,m_linkInertia[i],tmpMat3d);
	matTranspose(m_jntFrame[i].m_rot, Rt);
	matMultiply(tmpMat3d,Rt,inertia);
	
	// m*Jp'*Jp+Jo'*iner*Jo
	matTranspose(m_Jp[i],Jpt);
	matMultiply(Jpt,m_Jp[i], tmpMat7d);
	matMultiNum(tmpMat7d, m_linkMass[i],linkMassMat[i]);
	
	matTranspose(m_Jo[i],Jot);
	matMultiply(Jot,inertia, JotI);
	matMultiply(JotI,m_Jo[i],linkInerMat[i]);
END_FOR

// total mass mat
m_massMat :=g_zeroMat7d;
FOR i:=1 TO 9 DO
	matSelfAdd(m_massMat,linkMassMat[i]);
	matSelfAdd(m_massMat,linkInerMat[i]);
END_FOR

// add motor inertial 
FOR i:=1 TO 7 DO
	m_massMat[i,i]:=m_massMat[i,i]+m_motorInertia[i];
END_FOR

// mass mat inverse
invMat7(m_massMat,m_massMatInv);

// cartesian mass matrix
matTranspose(m_jaco, jacoT);
matMultiply(m_jaco,m_massMatInv, tmpMat67);
matMultiply(tmpMat67, jacoT, m_lambdaInv);
invMat6(m_lambdaInv, m_lambda);

// dyanmic nullspace
matMultiply(m_lambda, m_jaco, tmpMat67);
matMultiply(tmpMat67, m_massMatInv, m_JtGeneInv);
matMultiply(jacoT,m_JtGeneInv,tmpMat7d);
matSub(g_eye7d, tmpMat7d, m_dynaNullspace);
END_METHOD

// only update kinematic data
METHOD PROTECTED updateKinematic : BOOL
VAR_IN_OUT CONSTANT
	i_jntPos : Vec7d;
END_VAR
VAR
	Jp :ARRAY[1..3, 1..9] OF LREAL:=[27(0)];
	Jo :ARRAY[1..3, 1..9] OF LREAL:=[27(0)];
	jacoDH :Mat67;
	T :ST_Frame;
	i,j:INT;
	Pc,z,p:Vec3d;
	tcpPos :Vec3d;
	m,n :INT;
	
END_VAR
// tranform a joint positon to DH ones
m_armDH[1][4]:=i_jntPos[1];
m_armDH[2][4]:=i_jntPos[2];
m_armDH[3][4]:=i_jntPos[3]-i_jntPos[2];
m_armDH[4][4]:=i_jntPos[4]+i_jntPos[3]-i_jntPos[2]-pi/2;
m_armDH[5][4]:=i_jntPos[5];
m_armDH[6][4]:=i_jntPos[6];
m_armDH[7][4]:=i_jntPos[7];
m_armDH[8][4]:=i_jntPos[3];
m_armDH[9][4]:=i_jntPos[2]-i_jntPos[3];

// compute joint frame
m_jntFrame[1]:=DHTrans(m_armDH[1]);
T:=DHTrans(m_armDH[2]);
m_jntFrame[2]:=transform(m_jntFrame[1],T);
T:=DHTrans(m_armDH[3]);
m_jntFrame[3]:=transform(m_jntFrame[2],T);
T:=DHTrans(m_armDH[4]);
m_jntFrame[4]:=transform(m_jntFrame[3],T);
T:=DHTrans(m_armDH[5]);
m_jntFrame[5]:=transform(m_jntFrame[4],T);
T:=DHTrans(m_armDH[6]);
m_jntFrame[6]:=transform(m_jntFrame[5],T);
T:=DHTrans(m_armDH[7]);
m_jntFrame[7]:=transform(m_jntFrame[6],T);
T:=DHTrans(m_armDH[8]);
m_jntFrame[8]:=transform(m_jntFrame[1],T);
T:=DHTrans(m_armDH[9]);
m_jntFrame[9]:=transform(m_jntFrame[8],T);

// tcp jacobian
tcpPos:=m_jntFrame[7].m_pos;
FOR i:=1 TO 7 DO
	T:=m_jntFrame[i];
	z[1]:=T.m_rot[1,3];
	z[2]:=T.m_rot[2,3];
	z[3]:=T.m_rot[3,3];
	vecSub(tcpPos,T.m_pos,p);
	p:=cross(z,p);
	jacoDH[1,i]:=p[1];
	jacoDH[2,i]:=p[2];
	jacoDH[3,i]:=p[3];
	jacoDH[4,i]:=z[1];
	jacoDH[5,i]:=z[2];
	jacoDH[6,i]:=z[3];
END_FOR
// multiply m_jacoA
FOR m:=1 TO 6 DO 
	FOR n:=1 TO 7 DO
		IF 2=n THEN
			m_Jaco[m,n]:=jacoDH[m,2]-jacoDH[m,3]-jacoDH[m,4];
		ELSIF 3 =n THEN
			m_Jaco[m,n]:=jacoDH[m,3]+jacoDH[m,4];
		ELSE
			m_Jaco[m,n]:=jacoDH[m,n];
		END_IF
	END_FOR
END_FOR


// jacobian of mass center
FOR i:=1 TO 9 DO 
    T:=m_jntFrame[i];
	// mass center world position
    matMultiVec(T.m_rot,m_linkCOM[i], Pc);
	vecSelfAdd(Pc, T.m_pos);
    FOR j:=1 TO i DO
        IF (i>7 AND j>1 AND j<8) THEN
			Jp[1,j]:=0;
			Jp[2,j]:=0;
			Jp[3,j]:=0;
			Jo[1,j]:=0;
			Jo[2,j]:=0;
			Jo[3,j]:=0;
            CONTINUE;
        END_IF
        T:=m_jntFrame[j];
		z[1]:=T.m_rot[1,3];
		z[2]:=T.m_rot[2,3];
		z[3]:=T.m_rot[3,3];
        vecSub(Pc,T.m_pos,p);
		p:=cross(z,p);
		Jp[1,j]:=p[1];
		Jp[2,j]:=p[2];
		Jp[3,j]:=p[3];
        Jo[1,j]:=z[1];
		Jo[2,j]:=z[2];
		Jo[3,j]:=z[3];
    END_FOR
	// multiply m_jacoA
	FOR m:=1 TO 3 DO 
		FOR n:=1 TO 7 DO
			IF 2=n THEN
				m_Jp[i][m,n]:=Jp[m,2]-Jp[m,3]-Jp[m,4]+Jp[m,9];
				m_Jo[i][m,n]:=Jo[m,2]-Jo[m,3]-Jo[m,4]+Jo[m,9];
			ELSIF 3 =n THEN
				m_Jp[i][m,n]:=Jp[m,3]+Jp[m,4]+Jp[m,8]-Jp[m,9];
				m_Jo[i][m,n]:=Jo[m,3]+Jo[m,4]+Jo[m,8]-Jo[m,9];
			ELSE
				m_Jp[i][m,n]:=Jp[m,n];
				m_Jo[i][m,n]:=Jo[m,n];
			END_IF
		END_FOR
	END_FOR
END_FOR
END_METHOD

END_FUNCTION_BLOCK

// ---- AgiMaths/MatrixLib/matMultiNum.TcPOU
// matB=num*MatA
FUNCTION matMultiNum : BOOL
VAR_IN_OUT CONSTANT
	matA :ARRAY[*,*] OF LREAL;
	num : LREAL;
END_VAR

VAR_IN_OUT 
	matB :ARRAY[*,*] OF LREAL;
END_VAR

VAR
	m,n :DINT;
	i,j, k :DINT;
 
END_VAR

m:=UPPER_BOUND(matB,1);
n:= UPPER_BOUND(matB,2);
ASSERT(UPPER_BOUND(matA,1)=m);
ASSERT(UPPER_BOUND(matA,2)=n);

FOR i:=1 TO m DO
	FOR j:=1 TO n DO
		matB[i,j]:=num*matA[i,j];
	END_FOR
END_FOR

END_FUNCTION

// ---- AgiMaths/MatrixLib/matSelfAdd.TcPOU
// A +=B
FUNCTION matSelfAdd : BOOL
VAR_IN_OUT
	matA :ARRAY[*,*] OF LREAL;
END_VAR

VAR_IN_OUT CONSTANT
	matB :ARRAY[*,*] OF LREAL;
END_VAR

VAR
	m,n :DINT;
	i,j, k :DINT;
 
END_VAR

m:=UPPER_BOUND(matA,1);
n:= UPPER_BOUND(matA,2);
ASSERT(UPPER_BOUND(matB,1)=m);
ASSERT(UPPER_BOUND(matB,2)=n);
FOR i:=1 TO m DO
	FOR j:=1 TO n DO
		matA[i,j]:=matA[i,j]+matB[i,j];
	END_FOR
END_FOR

END_FUNCTION

// ---- AgiMaths/MatrixLib/invMat7.TcPOU
FUNCTION invMat7 : bool
VAR_IN_OUT CONSTANT
	mat :Mat7d;
END_VAR
VAR_IN_OUT
	invMat : Mat7d;
END_VAR
VAR
	n:INT:=7;
	m:INT:=1;
	b :ARRAY[1..7] OF LREAL := [7(0)];
	indxc,indxr, ipiv:ARRAY[1..7] OF INT := [7(0)];

	
	i,icol, irow, j,k,l,ll: INT;
	big, dum, pivinv,tmp: LREAL;
END_VAR

invMat := mat;
FOR i:=1 TO n DO   
    big:=0.0;
    FOR j:=1 TO n DO  
        IF (ipiv[j] <> 1) THEN
            FOR k:=1 TO n DO 
                IF (ipiv[k] = 0) THEN
                    IF (ABS(invMat[j,k]) >= big) THEN
                        big:=ABS(invMat[j,k]);
                        irow:=j;
                        icol:=k;
                    END_IF
                END_IF
            END_FOR
        END_IF
    END_FOR
    ipiv[icol]:=ipiv[icol]+1;
    
    IF (irow <> icol) THEN
        FOR l:=1 TO n DO 
            tmp:=invMat[irow,l];
            invMat[irow,l]:=invMat[icol,l];
            invMat[icol,l]:=tmp;
        END_FOR
 (*       FOR  l:=1 TO m DO  
            tmp:=b[irow,l];
            b[irow,l]:=b[icol,l];
            b[icol,l]:=tmp;
        END_FOR*)
    END_IF
	
    indxr[i]:=irow; 
    indxc[i]:=icol;
	
 	IF ABS(invMat[icol,icol]) < g_smallNum THEN 
          invMat7:=FALSE;
		  RETURN;
    END_IF
	
    pivinv:=1.0/invMat[icol,icol];
    invMat[icol,icol]:=1.0;
    FOR l:=1 TO n DO  
        invMat[icol,l] := invMat[icol,l]*pivinv;
    END_FOR
 (*   FOR l:=1 TO m DO 
        b[icol,l] := b[icol,l]*pivinv;
    END_FOR*)
    FOR ll:=1 TO n DO  
        IF (ll <> icol) THEN 
            dum:=invMat[ll,icol];
            invMat[ll,icol]:=0.0;
            FOR l:=1 TO n DO  
                invMat[ll,l]:=invMat[ll,l] - invMat[icol,l]*dum;
            END_FOR
   (*         FOR l:=1 TO m DO  
                b[ll,l]:=b[ll,l] - b[icol,l]*dum;
            END_FOR*)
        END_IF
    END_FOR

END_FOR


FOR l:=n-1 TO 1 BY -1 DO 
    IF (indxr[l] <> indxc[l]) THEN
        FOR k:=1 TO n DO
            tmp:=invMat[k,indxr[l]];
            invMat[k,indxr[l]]:=invMat[k,indxc[l]];
            invMat[k,indxc[l]]:=tmp;
        END_FOR
    END_IF
END_FOR

invMat7:=TRUE;

END_FUNCTION

// ---- AgiMaths/MatrixLib/invMat6.TcPOU
FUNCTION invMat6 : bool
VAR_IN_OUT CONSTANT
	mat :Mat6d;
END_VAR
VAR_IN_OUT
	invMat : Mat6d;
END_VAR
VAR
	n:INT:=6;
	m:INT:=1;
	b :ARRAY[1..6] OF LREAL := [6(0)];
	indxc,indxr, ipiv:ARRAY[1..6] OF INT := [6(0)];

	
	i,icol, irow, j,k,l,ll: INT;
	big, dum, pivinv,tmp: LREAL;
END_VAR

invMat := mat;
FOR i:=1 TO n DO   
    big:=0.0;
    FOR j:=1 TO n DO  
        IF (ipiv[j] <> 1) THEN
            FOR k:=1 TO n DO 
                IF (ipiv[k] = 0) THEN
                    IF (ABS(invMat[j,k]) >= big) THEN
                        big:=ABS(invMat[j,k]);
                        irow:=j;
                        icol:=k;
                    END_IF
                END_IF
            END_FOR
        END_IF
    END_FOR
    ipiv[icol]:=ipiv[icol]+1;
    
    IF (irow <> icol) THEN
        FOR l:=1 TO n DO 
            tmp:=invMat[irow,l];
            invMat[irow,l]:=invMat[icol,l];
            invMat[icol,l]:=tmp;
        END_FOR
 (*       FOR  l:=1 TO m DO  
            tmp:=b[irow,l];
            b[irow,l]:=b[icol,l];
            b[icol,l]:=tmp;
        END_FOR*)
    END_IF
	
    indxr[i]:=irow; 
    indxc[i]:=icol;
	
	IF ABS(invMat[icol,icol]) < g_smallNum THEN 
          invMat6:=FALSE;
		  RETURN;
    END_IF
	
    pivinv:=1.0/invMat[icol,icol];
    invMat[icol,icol]:=1.0;
    FOR l:=1 TO n DO  
        invMat[icol,l] := invMat[icol,l]*pivinv;
    END_FOR
 (*   FOR l:=1 TO m DO 
        b[icol,l] := b[icol,l]*pivinv;
    END_FOR*)
    FOR ll:=1 TO n DO  
        IF (ll <> icol) THEN 
            dum:=invMat[ll,icol];
            invMat[ll,icol]:=0.0;
            FOR l:=1 TO n DO  
                invMat[ll,l]:=invMat[ll,l] - invMat[icol,l]*dum;
            END_FOR
   (*         FOR l:=1 TO m DO  
                b[ll,l]:=b[ll,l] - b[icol,l]*dum;
            END_FOR*)
        END_IF
    END_FOR

END_FOR


FOR l:=n-1 TO 1 BY -1 DO 
    IF (indxr[l] <> indxc[l]) THEN
        FOR k:=1 TO n DO
            tmp:=invMat[k,indxr[l]];
            invMat[k,indxr[l]]:=invMat[k,indxc[l]];
            invMat[k,indxc[l]]:=tmp;
        END_FOR
    END_IF
END_FOR

invMat6:=TRUE;

END_FUNCTION

// ---- AgiMaths/MatrixLib/vecSelfAdd.TcPOU
// A +=B
FUNCTION vecSelfAdd : BOOL
VAR_IN_OUT
	vecA :ARRAY[*] OF LREAL;
END_VAR

VAR_IN_OUT CONSTANT
	vecB :ARRAY[*] OF LREAL;
END_VAR

VAR
	m,i :DINT;
 
END_VAR

m:=UPPER_BOUND(vecA,1);
ASSERT(UPPER_BOUND(VecB,1)=m);

FOR i:=1 TO m DO
		vecA[i]:=vecA[i]+vecB[i];
END_FOR

END_FUNCTION

// ---- FBs_RobotDynamics/FB_MasterFriciton.TcPOU
FUNCTION_BLOCK FB_MasterFriciton
VAR_INPUT
END_VAR
VAR_OUTPUT
END_VAR
VAR
	// joint friction compensation scale
	m_frictionCompScale :Vec7d :=[0, 0, 0, 0, 0.8, 0.4, 0];
	
	// joint velocity threshold for coulomb friction transition
	m_cFrictionVelThres : LREAL := 5.0 * g_deg2Rad;
	
	// arm index
	m_armIdx: INT ;
	
	// joint coulomb friction parameters: friction = a * gravityTrq + b;
	m_frictionParamA : Vec7d := g_zeroVec7d;
	m_frictionParamB : Vec7d := g_zeroVec7d;
	
	// joint damping
	m_jntDamp :Vec7d := g_zeroVec7d;
	
	// max joint friciton 
	m_maxFriction :Vec7d;
	

END_VAR

METHOD init : BOOL
VAR_INPUT
	i_armIdx :INT;
END_VAR
m_armIdx := i_armIdx;

m_frictionParamA := g_zeroVec7d;
m_frictionParamB := g_zeroVec7d;
m_jntDamp := g_zeroVec7d;
m_maxFriction := GVL_ArmDynamics.g_maxJntFriction;

m_frictionParamA[5] := GVL_ArmDynamics.g_jntFrictionParam[m_armIdx, 1];
m_frictionParamB[5] := GVL_ArmDynamics.g_jntFrictionParam[m_armIdx, 2];
m_frictionParamA[6] := GVL_ArmDynamics.g_jntFrictionParam[m_armIdx, 3];
m_frictionParamB[6] := GVL_ArmDynamics.g_jntFrictionParam[m_armIdx, 4];
END_METHOD

METHOD run : vec7d
VAR_IN_OUT CONSTANT
	// joint gravity torque
	i_jntGravity :Vec7d;
	
	// joint velocity
	i_jntVel :Vec7d;
END_VAR

VAR
	i:INT;
	transitScale:LREAL;
	cFriction, dFriction :LREAL;
END_VAR
FOR i:=1 TO g_mJntNum DO
	transitScale := LIMIT(0, ABS(i_jntVel[i]/m_cFrictionVelThres),1);
	cFriction:=m_frictionParamA[i]*ABS(i_jntGravity[i])+m_frictionParamB[i];
	cFriction:= transitScale * sign(i_jntVel[i]) * cFriction;
	
	dFriction:= i_jntVel[i] * m_jntDamp[i];
	
	run[i] := LIMIT(-m_maxFriction[i], m_frictionCompScale[i] * (cFriction+dFriction) ,m_maxFriction[i]);
END_FOR
END_METHOD

END_FUNCTION_BLOCK

// ---- FBs_Observer/FB_JntObserver.TcPOU
// joint state observer
// reference: Robotic Surgical System with Joint Motion Controller Adapted to Reduce Instrument Tip Vibration
FUNCTION_BLOCK FB_JntObserver
VAR_INPUT
END_VAR
VAR_OUTPUT
END_VAR
VAR
	// arm index
	m_armIdx :INT;
	
	// observer parameters
	m_L1,m_L2, m_L3:Vec7d;
	
	// joint parameters
	m_jntInertia, m_jntDamp : Vec7d;
	
	// joint observed status
	m_obvPos, m_obvVel, m_obvAcc, m_obvTrq :Vec7d;
END_VAR

METHOD PUBLIC init : BOOL
VAR_INPUT
	i_armIdx :INT;
	i_jntPos:Vec7d;
END_VAR
m_armIdx:=i_armIdx;

m_obvPos := i_jntPos;
m_obvVel := g_zeroVec7d;
m_obvAcc := g_zeroVec7d;
m_obvTrq := g_zeroVec7d;

m_L1 := g_jntObvParamL1;
m_L2 := g_jntObvParamL2;
m_L3 := g_jntObvParamL3;
m_jntDamp := g_jntObvDamp;
END_METHOD

METHOD PUBLIC run : vec7d
VAR_IN_OUT CONSTANT
	i_jntTrq :Vec7d;
	i_jntPos :Vec7d;
	i_massMat :Mat7d;
END_VAR

VAR 
	posErr :LREAL;
	i:INT;
END_VAR
FOR i:=1 TO g_mJntNum DO
	posErr := i_jntPos[i]-m_obvPos[i];
	
	m_obvTrq[i] := m_obvTrq[i]+g_armDynamicCycleTime*m_L3[i]*posErr;
	m_obvAcc[i] := (m_obvTrq[i] + i_jntTrq[i])/i_massMat[i,i];
	m_obvVel[i] := m_obvVel[i] + g_armDynamicCycleTime*(m_L2[i]*posErr + m_obvAcc[i] - m_obvVel[i]*m_jntDamp[i]/i_massMat[i,i])
					+ m_L1[i] * posErr;
	m_obvPos[i] := m_obvPos[i] + g_armDynamicCycleTime * m_obvVel[i];
END_FOR

run := m_obvTrq;
END_METHOD

END_FUNCTION_BLOCK

// ---- AgiMaths/Frames/invFrame.TcPOU
FUNCTION invFrame : ST_Frame
VAR_INPUT
	i_frame :ST_Frame;
END_VAR
VAR
	invPos :Vec3d;
END_VAR

matTranspose(i_frame.m_rot, invFrame.m_rot);
vecMultiNum(i_frame.m_pos, -1, invPos);
matMultiVec(invFrame.m_rot, invPos, invFrame.m_pos);

END_FUNCTION

// ---- AgiMaths/Frames/rotX.TcPOU
FUNCTION rotX : mat3d
VAR_INPUT
	i_ang : LREAL;
END_VAR
VAR
	rot :Mat3d := g_eye3d;
END_VAR

rot[2,2]:=COS(i_ang);
rot[3,3]:=rot[2,2];
rot[3,2]:=SIN(i_ang);
rot[2,3]:=-rot[3,2];
rotX :=rot;

END_FUNCTION

// ---- AgiMaths/Frames/rotZ.TcPOU
FUNCTION rotZ : mat3d
VAR_INPUT
	i_ang : LREAL;
END_VAR
VAR
	rot :Mat3d := g_eye3d;
END_VAR

rot[1,1]:=COS(i_ang);
rot[2,2]:=rot[1,1];
rot[2,1]:=SIN(i_ang);
rot[1,2]:=-rot[2,1];
rotZ:=rot;

END_FUNCTION

// ---- AgiMaths/MatrixLib/angAxis2Rot.TcPOU
FUNCTION angAxis2Rot : Mat3d
VAR_INPUT
	i_angle :LREAL;
	i_axis :Vec3d;
END_VAR
VAR
	cAng, sAng :LREAL;
	rx,ry,rz :LREAL;
END_VAR

IF norm(i_axis)<g_smallNum THEN
	angAxis2Rot := g_eye3d;
	RETURN;
END_IF

cAng :=COS(i_angle);
sAng := SIN(i_angle);
rx:=i_axis[1];
ry:=i_axis[2];
rz:=i_axis[3];

angAxis2Rot[1,1]:=rx*rx*(1-cAng)+cAng;
angAxis2Rot[2,1]:=rx*ry*(1-cAng)+rz*sAng;
angAxis2Rot[3,1]:=rx*rz*(1-cAng)-ry*sAng;

angAxis2Rot[1,2]:=rx*ry*(1-cAng)-rz*sAng;
angAxis2Rot[2,2]:=ry*ry*(1-cAng)+cAng;
angAxis2Rot[3,2]:=ry*rz*(1-cAng)+rx*sAng;

angAxis2Rot[1,3]:=rx*rz*(1-cAng)+ry*sAng;
angAxis2Rot[2,3]:=ry*rz*(1-cAng)-rx*sAng;
angAxis2Rot[3,3]:=rz*rz*(1-cAng)+cAng;

END_FUNCTION

// ---- AgiMaths/MatrixLib/Det5.TcPOU
FUNCTION Det5 : LREAL
VAR_IN_OUT CONSTANT
	mat: Mat5d;
END_VAR
VAR
	a11,a12,a13,a14,a15,a16:LREAL;
	a21,a22,a23,a24,a25,a26:LREAL;
	a31,a32,a33,a34,a35,a36:LREAL;
	a41,a42,a43,a44,a45,a46:LREAL;
	a51,a52,a53,a54,a55,a56:LREAL;
	a61,a62,a63,a64,a65,a66:LREAL;
END_VAR



//***************求取5X5矩阵的秩****************//
a11:=mat[1,1];
a12:=mat[1,2];
a13:=mat[1,3];
a14:=mat[1,4];
a15:=mat[1,5];

a21:=mat[2,1];
a22:=mat[2,2];
a23:=mat[2,3];
a24:=mat[2,4];
a25:=mat[2,5];

a31:=mat[3,1];
a32:=mat[3,2];
a33:=mat[3,3];
a34:=mat[3,4];
a35:=mat[3,5];

a41:=mat[4,1];
a42:=mat[4,2];
a43:=mat[4,3];
a44:=mat[4,4];
a45:=mat[4,5];

a51:=mat[5,1];
a52:=mat[5,2];
a53:=mat[5,3];
a54:=mat[5,4];
a55:=mat[5,5];

//Det5:=a11*a22*a33*a44*a55 - a11*a22*a33*a45*a54 - a11*a22*a34*a43*a55 + a11*a22*a34*a45*a53 + a11*a22*a35*a43*a54 - a11*a22*a35*a44*a53 - a11*a23*a32*a44*a55 + a11*a23*a32*a45*a54 + a11*a23*a34*a42*a55 - a11*a23*a34*a45*a52 - a11*a23*a35*a42*a54 + a11*a23*a35*a44*a52 + a11*a24*a32*a43*a55 - a11*a24*a32*a45*a53 - a11*a24*a33*a42*a55 + a11*a24*a33*a45*a52 + a11*a24*a35*a42*a53 - a11*a24*a35*a43*a52 - a11*a25*a32*a43*a54 + a11*a25*a32*a44*a53 + a11*a25*a33*a42*a54 - a11*a25*a33*a44*a52 - a11*a25*a34*a42*a53 + a11*a25*a34*a43*a52 - a12*a21*a33*a44*a55 + a12*a21*a33*a45*a54 + a12*a21*a34*a43*a55 - a12*a21*a34*a45*a53 - a12*a21*a35*a43*a54 + a12*a21*a35*a44*a53 + a12*a23*a31*a44*a55 - a12*a23*a31*a45*a54 - a12*a23*a34*a41*a55 + a12*a23*a34*a45*a51 + a12*a23*a35*a41*a54 - a12*a23*a35*a44*a51 - a12*a24*a31*a43*a55 + a12*a24*a31*a45*a53 + a12*a24*a33*a41*a55 - a12*a24*a33*a45*a51 - a12*a24*a35*a41*a53 + a12*a24*a35*a43*a51 + a12*a25*a31*a43*a54 - a12*a25*a31*a44*a53 - a12*a25*a33*a41*a54 + a12*a25*a33*a44*a51 + a12*a25*a34*a41*a53 - a12*a25*a34*a43*a51 + a13*a21*a32*a44*a55 - a13*a21*a32*a45*a54 - a13*a21*a34*a42*a55 + a13*a21*a34*a45*a52 + a13*a21*a35*a42*a54 - a13*a21*a35*a44*a52 - a13*a22*a31*a44*a55 + a13*a22*a31*a45*a54 + a13*a22*a34*a41*a55 - a13*a22*a34*a45*a51 - a13*a22*a35*a41*a54 + a13*a22*a35*a44*a51 + a13*a24*a31*a42*a55 - a13*a24*a31*a45*a52 - a13*a24*a32*a41*a55 + a13*a24*a32*a45*a51 + a13*a24*a35*a41*a52 - a13*a24*a35*a42*a51 - a13*a25*a31*a42*a54 + a13*a25*a31*a44*a52 + a13*a25*a32*a41*a54 - a13*a25*a32*a44*a51 - a13*a25*a34*a41*a52 + a13*a25*a34*a42*a51 - a14*a21*a32*a43*a55 + a14*a21*a32*a45*a53 + a14*a21*a33*a42*a55 - a14*a21*a33*a45*a52 - a14*a21*a35*a42*a53 + a14*a21*a35*a43*a52 + a14*a22*a31*a43*a55 - a14*a22*a31*a45*a53 - a14*a22*a33*a41*a55 + a14*a22*a33*a45*a51 + a14*a22*a35*a41*a53 - a14*a22*a35*a43*a51 - a14*a23*a31*a42*a55 + a14*a23*a31*a45*a52 + a14*a23*a32*a41*a55 - a14*a23*a32*a45*a51 - a14*a23*a35*a41*a52 + a14*a23*a35*a42*a51 + a14*a25*a31*a42*a53 - a14*a25*a31*a43*a52 - a14*a25*a32*a41*a53 + a14*a25*a32*a43*a51 + a14*a25*a33*a41*a52 - a14*a25*a33*a42*a51 + a15*a21*a32*a43*a54 - a15*a21*a32*a44*a53 - a15*a21*a33*a42*a54 + a15*a21*a33*a44*a52 + a15*a21*a34*a42*a53 - a15*a21*a34*a43*a52 - a15*a22*a31*a43*a54 + a15*a22*a31*a44*a53 + a15*a22*a33*a41*a54 - a15*a22*a33*a44*a51 - a15*a22*a34*a41*a53 + a15*a22*a34*a43*a51 + a15*a23*a31*a42*a54 - a15*a23*a31*a44*a52 - a15*a23*a32*a41*a54 + a15*a23*a32*a44*a51 + a15*a23*a34*a41*a52 - a15*a23*a34*a42*a51 - a15*a24*a31*a42*a53 + a15*a24*a31*a43*a52 + a15*a24*a32*a41*a53 - a15*a24*a32*a43*a51 - a15*a24*a33*a41*a52 + a15*a24*a33*a42*a51;
Det5:=((a31*a43*a52 - a31*a42*a53 + a32*a41*a53 - a32*a43*a51 - a33*a41*a52 + a33*a42*a51)*a24 + (a31*a42*a54 - a31*a44*a52 - a32*a41*a54 + a32*a44*a51 + a34*a41*a52 - a34*a42*a51)*a23 + (a31*a44*a53 - a31*a43*a54 + a33*a41*a54 - a33*a44*a51 - a34*a41*a53 + a34*a43*a51)*a22 + (a32*a43*a54 - a32*a44*a53 - a33*a42*a54 + a33*a44*a52 + a34*a42*a53 - a34*a43*a52)*a21)*a15 
	+ ((a31*a42*a53 - a31*a43*a52 - a32*a41*a53 + a32*a43*a51 + a33*a41*a52 - a33*a42*a51)*a25 + (a31*a45*a52 - a31*a42*a55 + a32*a41*a55 - a32*a45*a51 - a35*a41*a52 + a35*a42*a51)*a23 + (a31*a43*a55 - a31*a45*a53 - a33*a41*a55 + a33*a45*a51 + a35*a41*a53 - a35*a43*a51)*a22 + (a32*a45*a53 - a32*a43*a55 + a33*a42*a55 - a33*a45*a52 - a35*a42*a53 + a35*a43*a52)*a21)*a14 
	+ ((a31*a44*a52 - a31*a42*a54 + a32*a41*a54 - a32*a44*a51 - a34*a41*a52 + a34*a42*a51)*a25 + (a31*a42*a55 - a31*a45*a52 - a32*a41*a55 + a32*a45*a51 + a35*a41*a52 - a35*a42*a51)*a24 + (a31*a45*a54 - a31*a44*a55 + a34*a41*a55 - a34*a45*a51 - a35*a41*a54 + a35*a44*a51)*a22 + (a32*a44*a55 - a32*a45*a54 - a34*a42*a55 + a34*a45*a52 + a35*a42*a54 - a35*a44*a52)*a21)*a13 
	+ ((a31*a43*a54 - a31*a44*a53 - a33*a41*a54 + a33*a44*a51 + a34*a41*a53 - a34*a43*a51)*a25 + (a31*a45*a53 - a31*a43*a55 + a33*a41*a55 - a33*a45*a51 - a35*a41*a53 + a35*a43*a51)*a24 + (a31*a44*a55 - a31*a45*a54 - a34*a41*a55 + a34*a45*a51 + a35*a41*a54 - a35*a44*a51)*a23 + (a33*a45*a54 - a33*a44*a55 + a34*a43*a55 - a34*a45*a53 - a35*a43*a54 + a35*a44*a53)*a21)*a12 
	+ ((a32*a44*a53 - a32*a43*a54 + a33*a42*a54 - a33*a44*a52 - a34*a42*a53 + a34*a43*a52)*a25 + (a32*a43*a55 - a32*a45*a53 - a33*a42*a55 + a33*a45*a52 + a35*a42*a53 - a35*a43*a52)*a24 + (a32*a45*a54 - a32*a44*a55 + a34*a42*a55 - a34*a45*a52 - a35*a42*a54 + a35*a44*a52)*a23 + (a33*a44*a55 - a33*a45*a54 - a34*a43*a55 + a34*a45*a53 + a35*a43*a54 - a35*a44*a53)*a22)*a11;

END_FUNCTION

// ---- AgiMaths/MatrixLib/Det6.TcPOU
FUNCTION Det6 : LREAL
VAR_IN_OUT CONSTANT
	mat: Mat6d;
END_VAR
VAR
	a11,a12,a13,a14,a15,a16:LREAL;
	a21,a22,a23,a24,a25,a26:LREAL;
	a31,a32,a33,a34,a35,a36:LREAL;
	a41,a42,a43,a44,a45,a46:LREAL;
	a51,a52,a53,a54,a55,a56:LREAL;
	a61,a62,a63,a64,a65,a66:LREAL;
END_VAR


a11:=mat[1,1];
a12:=mat[1,2];
a13:=mat[1,3];
a14:=mat[1,4];
a15:=mat[1,5];
a16:=mat[1,6];

a21:=mat[2,1];
a22:=mat[2,2];
a23:=mat[2,3];
a24:=mat[2,4];
a25:=mat[2,5];
a26:=mat[2,6];

a31:=mat[3,1];
a32:=mat[3,2];
a33:=mat[3,3];
a34:=mat[3,4];
a35:=mat[3,5];
a36:=mat[3,6];

a41:=mat[4,1];
a42:=mat[4,2];
a43:=mat[4,3];
a44:=mat[4,4];
a45:=mat[4,5];
a46:=mat[4,6];

a51:=mat[5,1];
a52:=mat[5,2];
a53:=mat[5,3];
a54:=mat[5,4];
a55:=mat[5,5];
a56:=mat[5,6];

a61:=mat[6,1];
a62:=mat[6,2];
a63:=mat[6,3];
a64:=mat[6,4];
a65:=mat[6,5];
a66:=mat[6,6];

